LIN {X 0,Y 312.695,Z 496.66,A -85,B 0,C 180,E1 -15735.686,E2 -15735.686} C_VEL
LIN {X 0,Y 312.703,Z 496.659,A -85,B 0,C 180,E1 -15739.642,E2 -15739.642} C_VEL
LIN {X 0,Y 312.873,Z 496.634,A -85,B 0,C 180,E1 -15742.254,E2 -15742.254} C_VEL
LIN {X 0,Y 312.72,Z 496.654,A -85,B 0,C 180,E1 -15744.842,E2 -15744.842} C_VEL
LIN {X 0,Y 312.954,Z 496.629,A -85,B 0,C 180,E1 -15747.426,E2 -15747.426} C_VEL
LIN {X 0,Y 313.122,Z 496.604,A -85,B 0,C 180,E1 -15750,E2 -15750} C_VEL
LIN {X 0,Y 312.94,Z 496.626,A -85,B 0,C 180,E1 -15752.574,E2 -15752.574} C_VEL
LIN {X 0,Y 312.911,Z 496.629,A -85,B 0,C 180,E1 -15756.448,E2 -15756.448} C_VEL
LIN {X 0,Y 312.789,Z 496.646,A -85,B 0,C 180,E1 -15759.049,E2 -15759.049} C_VEL
LIN {X 0,Y 312.636,Z 496.666,A -85,B 0,C 180,E1 -15762.991,E2 -15762.991} C_VEL
LIN {X 0,Y 312.639,Z 496.666,A -85,B 0,C 180,E1 -15765.65,E2 -15765.65} C_VEL
LIN {X 0,Y 312.631,Z 496.668,A -85,B 0,C 180,E1 -15769.237,E2 -15769.237} C_VEL
LIN {X 0,Y 312.547,Z 496.676,A -85,B 0,C 180,E1 -15772.789,E2 -15772.789} C_VEL
LIN {X 0,Y 312.598,Z 496.669,A -85,B 0,C 180,E1 -15775.933,E2 -15775.933} C_VEL
LIN {X 0,Y 312.539,Z 496.679,A -85,B 0,C 180,E1 -15779.651,E2 -15779.651} C_VEL
LIN {X 0,Y 312.52,Z 496.68,A -85,B 0,C 180,E1 -15783.689,E2 -15783.689} C_VEL
LIN {X 0,Y 312.539,Z 496.681,A -85,B 0,C 180,E1 -15787.383,E2 -15787.383} C_VEL
LIN {X 0,Y 312.491,Z 496.682,A -85,B 0,C 180,E1 -15790.709,E2 -15790.709} C_VEL
LIN {X 0,Y 312.473,Z 496.684,A -85,B 0,C 180,E1 -15794.206,E2 -15794.206} C_VEL
LIN {X 0,Y 312.487,Z 496.683,A -85,B 0,C 180,E1 -15797.918,E2 -15797.918} C_VEL
LIN {X 0,Y 312.507,Z 496.681,A -85,B 0,C 180,E1 -15801.917,E2 -15801.917} C_VEL
LIN {X 0,Y 312.533,Z 496.677,A -85,B 0,C 180,E1 -15804.22,E2 -15804.22} C_VEL
LIN {X 0,Y 312.548,Z 496.702,A -85,B 0,C 180,E1 -15806.423,E2 -15806.423} C_VEL
LIN {X 0,Y 316.105,Z 512.177,A -85,B 0,C 180,E1 -15809.735,E2 -15809.735} C_VEL
LIN {X 0,Y 318.578,Z 524.112,A -85,B 0,C 180,E1 -15812.214,E2 -15812.214} C_VEL
LIN {X 0,Y 317.779,Z 535.92,A -85,B 0,C 180,E1 -15814.452,E2 -15814.452} C_VEL
LIN {X 0,Y 317.727,Z 536.622,A -85,B 0,C 180,E1 -15814.586,E2 -15814.586} C_VEL
LIN {X 0,Y 316.838,Z 539.658,A -85,B 0,C 180,E1 -15815.123,E2 -15815.123} C_VEL
LIN {X 0,Y 313.587,Z 544.619,A -85,B 0,C 180,E1 -15815.91,E2 -15815.91} C_VEL
LIN {X 0,Y 310.704,Z 549.223,A -85,B 0,C 180,E1 -15816.517,E2 -15816.517} C_VEL
LIN {X 0,Y 310.133,Z 552.013,A -85,B 0,C 180,E1 -15816.724,E2 -15816.724} C_VEL
LIN {X 0,Y 310.154,Z 552.609,A -85,B 0,C 180,E1 -15816.751,E2 -15816.751} C_VEL
LIN {X 0,Y 313.108,Z 577.851,A -85,B 0,C 180,E1 -15817.752,E2 -15817.752} C_VEL
LIN {X 0,Y 310.286,Z 660.865,A -85,B 0,C 180,E1 -15820.483,E2 -15820.483} C_VEL
LIN {X 0,Y 309.628,Z 673.725,A -85,B 0,C 180,E1 -15821.128,E2 -15821.128} C_VEL
LIN {X 0,Y 308.833,Z 687.47,A -85,B 0,C 180,E1 -15822.109,E2 -15822.109} C_VEL
LIN {X 0,Y 308,Z 699.244,A -85,B 0,C 180,E1 -15823.207,E2 -15823.207} C_VEL
LIN {X 0,Y 307.266,Z 709.548,A -85,B 0,C 180,E1 -15824.41,E2 -15824.41} C_VEL
LIN {X 0,Y 306.424,Z 719.942,A -85,B 0,C 180,E1 -15825.896,E2 -15825.896} C_VEL
LIN {X 0,Y 305.623,Z 728.532,A -85,B 0,C 180,E1 -15827.381,E2 -15827.381} C_VEL
LIN {X 0,Y 304.853,Z 737.882,A -85,B 0,C 180,E1 -15829.372,E2 -15829.372} C_VEL
LIN {X 0,Y 304.29,Z 745.423,A -85,B 0,C 180,E1 -15831.366,E2 -15831.366} C_VEL
LIN {X 0,Y 303.987,Z 751.404,A -85,B 0,C 180,E1 -15833.362,E2 -15833.362} C_VEL
LIN {X 0,Y 303.777,Z 756.071,A -85,B 0,C 180,E1 -15835.355,E2 -15835.355} C_VEL
LIN {X 0,Y 303.663,Z 759.57,A -85,B 0,C 180,E1 -15837.347,E2 -15837.347} C_VEL
LIN {X 0,Y 303.58,Z 761.313,A -85,B 0,C 180,E1 -15838.673,E2 -15838.673} C_VEL
LIN {X 0,Y 303.601,Z 762.593,A -85,B 0,C 180,E1 -15840,E2 -15840} C_VEL
LIN {X 0,Y 303.634,Z 763.4,A -85,B 0,C 180,E1 -15841.326,E2 -15841.326} C_VEL
LIN {X 0,Y 303.73,Z 763.791,A -85,B 0,C 180,E1 -15842.653,E2 -15842.653} C_VEL
LIN {X 0,Y 303.896,Z 763.755,A -85,B 0,C 180,E1 -15843.978,E2 -15843.978} C_VEL
LIN {X 0,Y 304.174,Z 763.245,A -85,B 0,C 180,E1 -15845.303,E2 -15845.303} C_VEL
LIN {X 0,Y 304.765,Z 761.541,A -85,B 0,C 180,E1 -15847.432,E2 -15847.432} C_VEL
LIN {X 0,Y 305.648,Z 758.098,A -85,B 0,C 180,E1 -15849.931,E2 -15849.931} C_VEL
LIN {X 0,Y 306.73,Z 754.162,A -85,B 0,C 180,E1 -15851.901,E2 -15851.901} C_VEL
LIN {X 0,Y 308.02,Z 749.044,A -85,B 0,C 180,E1 -15853.862,E2 -15853.862} C_VEL
LIN {X 0,Y 309.69,Z 742.568,A -85,B 0,C 180,E1 -15855.803,E2 -15855.803} C_VEL
LIN {X 0,Y 311.786,Z 734.624,A -85,B 0,C 180,E1 -15857.716,E2 -15857.716} C_VEL
LIN {X 0,Y 313.755,Z 726.562,A -85,B 0,C 180,E1 -15859.293,E2 -15859.293} C_VEL
LIN {X 0,Y 316.124,Z 715.871,A -85,B 0,C 180,E1 -15860.975,E2 -15860.975} C_VEL
LIN {X 0,Y 318.27,Z 704.858,A -85,B 0,C 180,E1 -15862.39,E2 -15862.39} C_VEL
LIN {X 0,Y 320.467,Z 692.846,A -85,B 0,C 180,E1 -15863.593,E2 -15863.593} C_VEL
LIN {X 0,Y 322.376,Z 680.473,A -85,B 0,C 180,E1 -15864.556,E2 -15864.556} C_VEL
LIN {X 0,Y 324.061,Z 666.63,A -85,B 0,C 180,E1 -15865.361,E2 -15865.361} C_VEL
LIN {X 0,Y 326.296,Z 642.291,A -85,B 0,C 180,E1 -15866.332,E2 -15866.332} C_VEL
LIN {X 0,Y 332.02,Z 585.244,A -85,B 0,C 180,E1 -15868.52,E2 -15868.52} C_VEL
LIN {X 0,Y 330.422,Z 572.445,A -85,B 0,C 180,E1 -15869.651,E2 -15869.651} C_VEL
LIN {X 0,Y 328.053,Z 558.26,A -85,B 0,C 180,E1 -15871.202,E2 -15871.202} C_VEL
LIN {X 0,Y 327.111,Z 552.951,A -85,B 0,C 180,E1 -15871.875,E2 -15871.875} C_VEL
LIN {X 0,Y 326.796,Z 547.751,A -85,B 0,C 180,E1 -15873.522,E2 -15873.522} C_VEL
LIN {X 0,Y 326.075,Z 542.207,A -85,B 0,C 180,E1 -15875.587,E2 -15875.587} C_VEL
LIN {X 0,Y 325.136,Z 537.325,A -85,B 0,C 180,E1 -15877.875,E2 -15877.875} C_VEL
LIN {X 0,Y 324.526,Z 534.263,A -85,B 0,C 180,E1 -15879.638,E2 -15879.638} C_VEL
LIN {X 0,Y 323.75,Z 531.075,A -85,B 0,C 180,E1 -15882.295,E2 -15882.295} C_VEL
LIN {X 0,Y 323.483,Z 529.687,A -85,B 0,C 180,E1 -15884.196,E2 -15884.196} C_VEL
LIN {X 0,Y 323.536,Z 529.08,A -85,B 0,C 180,E1 -15885.963,E2 -15885.963} C_VEL
LIN {X 0,Y 323.915,Z 529.107,A -85,B 0,C 180,E1 -15887.731,E2 -15887.731} C_VEL
LIN {X 0,Y 324.623,Z 529.847,A -85,B 0,C 180,E1 -15889.497,E2 -15889.497} C_VEL
LIN {X 0,Y 325.763,Z 531.237,A -85,B 0,C 180,E1 -15891.27,E2 -15891.27} C_VEL
LIN {X 0,Y 327.409,Z 533.393,A -85,B 0,C 180,E1 -15893.056,E2 -15893.056} C_VEL
LIN {X 0,Y 329.137,Z 536.699,A -85,B 0,C 180,E1 -15894.793,E2 -15894.793} C_VEL
LIN {X 0,Y 329.649,Z 540.65,A -85,B 0,C 180,E1 -15895.886,E2 -15895.886} C_VEL
LIN {X 0,Y 330.931,Z 549.612,A -85,B 0,C 180,E1 -15897.932,E2 -15897.932} C_VEL
LIN {X 0,Y 331.047,Z 551.894,A -85,B 0,C 180,E1 -15898.332,E2 -15898.332} C_VEL
LIN {X 0,Y 330.217,Z 558.252,A -85,B 0,C 180,E1 -15899.044,E2 -15899.044} C_VEL
LIN {X 0,Y 330.357,Z 566.805,A -85,B 0,C 180,E1 -15899.668,E2 -15899.668} C_VEL
LIN {X 0,Y 321.228,Z 657.87,A -85,B 0,C 180,E1 -15903.396,E2 -15903.396} C_VEL
LIN {X 0,Y 319.332,Z 680.325,A -85,B 0,C 180,E1 -15904.367,E2 -15904.367} C_VEL
LIN {X 0,Y 317.783,Z 694.511,A -85,B 0,C 180,E1 -15905.267,E2 -15905.267} C_VEL
LIN {X 0,Y 316.222,Z 706.55,A -85,B 0,C 180,E1 -15906.266,E2 -15906.266} C_VEL
LIN {X 0,Y 314.48,Z 718.218,A -85,B 0,C 180,E1 -15907.498,E2 -15907.498} C_VEL
LIN {X 0,Y 312.297,Z 730.334,A -85,B 0,C 180,E1 -15909.068,E2 -15909.068} C_VEL
LIN {X 0,Y 310.283,Z 741.053,A -85,B 0,C 180,E1 -15910.826,E2 -15910.826} C_VEL
LIN {X 0,Y 308.438,Z 750.629,A -85,B 0,C 180,E1 -15912.77,E2 -15912.77} C_VEL
LIN {X 0,Y 306.979,Z 758.385,A -85,B 0,C 180,E1 -15914.735,E2 -15914.735} C_VEL
LIN {X 0,Y 305.773,Z 764.7,A -85,B 0,C 180,E1 -15916.712,E2 -15916.712} C_VEL
LIN {X 0,Y 304.895,Z 769.78,A -85,B 0,C 180,E1 -15918.701,E2 -15918.701} C_VEL
LIN {X 0,Y 304.243,Z 773.698,A -85,B 0,C 180,E1 -15920.694,E2 -15920.694} C_VEL
LIN {X 0,Y 303.964,Z 775.739,A -85,B 0,C 180,E1 -15922.026,E2 -15922.026} C_VEL
LIN {X 0,Y 303.689,Z 778.175,A -85,B 0,C 180,E1 -15924.332,E2 -15924.332} C_VEL
LIN {X 0,Y 303.601,Z 779.137,A -85,B 0,C 180,E1 -15926.018,E2 -15926.018} C_VEL
LIN {X 0,Y 303.627,Z 779.384,A -85,B 0,C 180,E1 -15927.347,E2 -15927.347} C_VEL
LIN {X 0,Y 303.622,Z 779.172,A -85,B 0,C 180,E1 -15928.674,E2 -15928.674} C_VEL
LIN {X 0,Y 303.591,Z 780.184,A -85,B 0,C 180,E1 -15931.327,E2 -15931.327} C_VEL
LIN {X 0,Y 303.608,Z 780.324,A -85,B 0,C 180,E1 -15932.654,E2 -15932.654} C_VEL
LIN {X 0,Y 303.617,Z 779.456,A -85,B 0,C 180,E1 -15935.313,E2 -15935.313} C_VEL
LIN {X 0,Y 303.931,Z 777.116,A -85,B 0,C 180,E1 -15937.975,E2 -15937.975} C_VEL
LIN {X 0,Y 304.585,Z 773.291,A -85,B 0,C 180,E1 -15940.638,E2 -15940.638} C_VEL
LIN {X 0,Y 305.761,Z 767.896,A -85,B 0,C 180,E1 -15943.289,E2 -15943.289} C_VEL
LIN {X 0,Y 306.969,Z 762.706,A -85,B 0,C 180,E1 -15945.266,E2 -15945.266} C_VEL
LIN {X 0,Y 308.805,Z 755.301,A -85,B 0,C 180,E1 -15947.551,E2 -15947.551} C_VEL
LIN {X 0,Y 311.045,Z 746.197,A -85,B 0,C 180,E1 -15949.811,E2 -15949.811} C_VEL
LIN {X 0,Y 313.455,Z 736.695,A -85,B 0,C 180,E1 -15951.713,E2 -15951.713} C_VEL
LIN {X 0,Y 316.278,Z 725.263,A -85,B 0,C 180,E1 -15953.577,E2 -15953.577} C_VEL
LIN {X 0,Y 318.903,Z 713.895,A -85,B 0,C 180,E1 -15955.088,E2 -15955.088} C_VEL
LIN {X 0,Y 321.678,Z 700.835,A -85,B 0,C 180,E1 -15956.481,E2 -15956.481} C_VEL
LIN {X 0,Y 324.109,Z 687.483,A -85,B 0,C 180,E1 -15957.613,E2 -15957.613} C_VEL
LIN {X 0,Y 326.649,Z 671.83,A -85,B 0,C 180,E1 -15958.602,E2 -15958.602} C_VEL
LIN {X 0,Y 328.391,Z 657.161,A -85,B 0,C 180,E1 -15959.268,E2 -15959.268} C_VEL
LIN {X 0,Y 335.537,Z 586.231,A -85,B 0,C 180,E1 -15961.806,E2 -15961.806} C_VEL
LIN {X 0,Y 337.662,Z 566.7,A -85,B 0,C 180,E1 -15962.538,E2 -15962.538} C_VEL
LIN {X 0,Y 337.163,Z 562,A -85,B 0,C 180,E1 -15962.964,E2 -15962.964} C_VEL
LIN {X 0,Y 334.12,Z 555.825,A -85,B 0,C 180,E1 -15964.156,E2 -15964.156} C_VEL
LIN {X 0,Y 331.829,Z 551.509,A -85,B 0,C 180,E1 -15965.145,E2 -15965.145} C_VEL
LIN {X 0,Y 329.918,Z 548.193,A -85,B 0,C 180,E1 -15966.033,E2 -15966.033} C_VEL
LIN {X 0,Y 327.363,Z 544.086,A -85,B 0,C 180,E1 -15967.336,E2 -15967.336} C_VEL
LIN {X 0,Y 323.847,Z 539.068,A -85,B 0,C 180,E1 -15969.498,E2 -15969.498} C_VEL
LIN {X 0,Y 320.513,Z 534.919,A -85,B 0,C 180,E1 -15972.459,E2 -15972.459} C_VEL
LIN {X 0,Y 319.82,Z 533.854,A -85,B 0,C 180,E1 -15973.517,E2 -15973.517} C_VEL
LIN {X 0,Y 319.684,Z 533.495,A -85,B 0,C 180,E1 -15976.509,E2 -15976.509} C_VEL
LIN {X 0,Y 319.826,Z 534.162,A -85,B 0,C 180,E1 -15978.759,E2 -15978.759} C_VEL
LIN {X 0,Y 320.214,Z 535.661,A -85,B 0,C 180,E1 -15980.843,E2 -15980.843} C_VEL
LIN {X 0,Y 323.301,Z 540.989,A -85,B 0,C 180,E1 -15983.922,E2 -15983.922} C_VEL
LIN {X 0,Y 324.67,Z 543.01,A -85,B 0,C 180,E1 -15984.879,E2 -15984.879} C_VEL
LIN {X 0,Y 328.101,Z 549.368,A -85,B 0,C 180,E1 -15986.957,E2 -15986.957} C_VEL
LIN {X 0,Y 330.938,Z 555.184,A -85,B 0,C 180,E1 -15988.434,E2 -15988.434} C_VEL
LIN {X 0,Y 332.724,Z 559.305,A -85,B 0,C 180,E1 -15989.287,E2 -15989.287} C_VEL
LIN {X 0,Y 334.38,Z 571.019,A -85,B 0,C 180,E1 -15990.609,E2 -15990.609} C_VEL
LIN {X 0,Y 335.309,Z 581.125,A -85,B 0,C 180,E1 -15991.553,E2 -15991.553} C_VEL
LIN {X 0,Y 335.436,Z 584.56,A -85,B 0,C 180,E1 -15991.807,E2 -15991.807} C_VEL
LIN {X 0,Y 326.755,Z 659.896,A -85,B 0,C 180,E1 -15994.864,E2 -15994.864} C_VEL
LIN {X 0,Y 324.963,Z 672.654,A -85,B 0,C 180,E1 -15995.61,E2 -15995.61} C_VEL
LIN {X 0,Y 322.419,Z 687.269,A -85,B 0,C 180,E1 -15996.747,E2 -15996.747} C_VEL
LIN {X 0,Y 320.224,Z 699.057,A -85,B 0,C 180,E1 -15997.923,E2 -15997.923} C_VEL
LIN {X 0,Y 317.517,Z 711.185,A -85,B 0,C 180,E1 -15999.428,E2 -15999.428} C_VEL
LIN {X 0,Y 314.904,Z 722.101,A -85,B 0,C 180,E1 -16001.119,E2 -16001.119} C_VEL
LIN {X 0,Y 312.39,Z 731.847,A -85,B 0,C 180,E1 -16002.994,E2 -16002.994} C_VEL
LIN {X 0,Y 310.347,Z 739.777,A -85,B 0,C 180,E1 -16004.905,E2 -16004.905} C_VEL
LIN {X 0,Y 308.598,Z 746.288,A -85,B 0,C 180,E1 -16006.836,E2 -16006.836} C_VEL
LIN {X 0,Y 307.089,Z 751.53,A -85,B 0,C 180,E1 -16008.783,E2 -16008.783} C_VEL
LIN {X 0,Y 305.999,Z 755.591,A -85,B 0,C 180,E1 -16010.748,E2 -16010.748} C_VEL
LIN {X 0,Y 305.368,Z 757.72,A -85,B 0,C 180,E1 -16012.063,E2 -16012.063} C_VEL
LIN {X 0,Y 304.764,Z 759.412,A -85,B 0,C 180,E1 -16013.379,E2 -16013.379} C_VEL
LIN {X 0,Y 304.373,Z 760.671,A -85,B 0,C 180,E1 -16014.701,E2 -16014.701} C_VEL
LIN {X 0,Y 304.136,Z 761.512,A -85,B 0,C 180,E1 -16016.025,E2 -16016.025} C_VEL
LIN {X 0,Y 303.912,Z 761.908,A -85,B 0,C 180,E1 -16017.349,E2 -16017.349} C_VEL
LIN {X 0,Y 303.732,Z 761.869,A -85,B 0,C 180,E1 -16018.674,E2 -16018.674} C_VEL
LIN {X 0,Y 303.639,Z 761.416,A -85,B 0,C 180,E1 -16020,E2 -16020} C_VEL
LIN {X 0,Y 303.615,Z 760.545,A -85,B 0,C 180,E1 -16021.326,E2 -16021.326} C_VEL
LIN {X 0,Y 303.658,Z 759.214,A -85,B 0,C 180,E1 -16022.653,E2 -16022.653} C_VEL
LIN {X 0,Y 303.667,Z 756.37,A -85,B 0,C 180,E1 -16024.646,E2 -16024.646} C_VEL
LIN {X 0,Y 303.858,Z 752.437,A -85,B 0,C 180,E1 -16026.641,E2 -16026.641} C_VEL
LIN {X 0,Y 304.142,Z 747.299,A -85,B 0,C 180,E1 -16028.638,E2 -16028.638} C_VEL
LIN {X 0,Y 304.695,Z 739.609,A -85,B 0,C 180,E1 -16030.97,E2 -16030.97} C_VEL
LIN {X 0,Y 305.417,Z 731.304,A -85,B 0,C 180,E1 -16032.965,E2 -16032.965} C_VEL
LIN {X 0,Y 306.216,Z 721.523,A -85,B 0,C 180,E1 -16034.853,E2 -16034.853} C_VEL
LIN {X 0,Y 307.126,Z 711.43,A -85,B 0,C 180,E1 -16036.45,E2 -16036.45} C_VEL
LIN {X 0,Y 308.19,Z 699.881,A -85,B 0,C 180,E1 -16037.93,E2 -16037.93} C_VEL
LIN {X 0,Y 309.268,Z 687.138,A -85,B 0,C 180,E1 -16039.239,E2 -16039.239} C_VEL
LIN {X 0,Y 310.192,Z 673.757,A -85,B 0,C 180,E1 -16040.3,E2 -16040.3} C_VEL
LIN {X 0,Y 311.018,Z 659.239,A -85,B 0,C 180,E1 -16041.152,E2 -16041.152} C_VEL
LIN {X 0,Y 311.791,Z 641.246,A -85,B 0,C 180,E1 -16041.834,E2 -16041.834} C_VEL
LIN {X 0,Y 314.384,Z 574.76,A -85,B 0,C 180,E1 -16044.078,E2 -16044.078} C_VEL
LIN {X 0,Y 310.271,Z 540.944,A -85,B 0,C 180,E1 -16045.514,E2 -16045.514} C_VEL
LIN {X 0,Y 310.116,Z 539.007,A -85,B 0,C 180,E1 -16045.595,E2 -16045.595} C_VEL
LIN {X 0,Y 311.695,Z 526.352,A -85,B 0,C 180,E1 -16048.628,E2 -16048.628} C_VEL
LIN {X 0,Y 309.2,Z 514.335,A -85,B 0,C 180,E1 -16051.833,E2 -16051.833} C_VEL
LIN {X 0,Y 306.408,Z 501.538,A -85,B 0,C 180,E1 -16055.391,E2 -16055.391} C_VEL
LIN {X 0,Y 305.508,Z 497.552,A -85,B 0,C 180,E1 -16056.557,E2 -16056.557} C_VEL
LIN {X 0,Y 305.46,Z 497.558,A -85,B 0,C 180,E1 -16060.107,E2 -16060.107} C_VEL
LIN {X 0,Y 305.43,Z 497.566,A -85,B 0,C 180,E1 -16063.654,E2 -16063.654} C_VEL
LIN {X 0,Y 305.456,Z 497.562,A -85,B 0,C 180,E1 -16067.414,E2 -16067.414} C_VEL
LIN {X 0,Y 305.477,Z 497.561,A -85,B 0,C 180,E1 -16071.597,E2 -16071.597} C_VEL
LIN {X 0,Y 305.464,Z 497.557,A -85,B 0,C 180,E1 -16074.887,E2 -16074.887} C_VEL
LIN {X 0,Y 305.454,Z 497.558,A -85,B 0,C 180,E1 -16078.354,E2 -16078.354} C_VEL
LIN {X 0,Y 305.522,Z 497.552,A -85,B 0,C 180,E1 -16081.114,E2 -16081.114} C_VEL
LIN {X 0,Y 305.573,Z 497.544,A -85,B 0,C 180,E1 -16084.088,E2 -16084.088} C_VEL
LIN {X 0,Y 305.503,Z 497.552,A -85,B 0,C 180,E1 -16088.403,E2 -16088.403} C_VEL
LIN {X 0,Y 305.592,Z 497.544,A -85,B 0,C 180,E1 -16091.218,E2 -16091.218} C_VEL
LIN {X 0,Y 305.65,Z 497.538,A -85,B 0,C 180,E1 -16095.349,E2 -16095.349} C_VEL
LIN {X 0,Y 305.64,Z 497.54,A -85,B 0,C 180,E1 -16099.4,E2 -16099.4} C_VEL
LIN {X 0,Y 305.814,Z 497.514,A -85,B 0,C 180,E1 -16102.074,E2 -16102.074} C_VEL
LIN {X 0,Y 305.692,Z 497.529,A -85,B 0,C 180,E1 -16104.723,E2 -16104.723} C_VEL
LIN {X 0,Y 305.961,Z 497.495,A -85,B 0,C 180,E1 -16108.684,E2 -16108.684} C_VEL
LIN {X 0,Y 305.959,Z 497.499,A -85,B 0,C 180,E1 -16111.316,E2 -16111.316} C_VEL
LIN {X 0,Y 305.853,Z 497.508,A -85,B 0,C 180,E1 -16116.597,E2 -16116.597} C_VEL
LIN {X 0,Y 305.737,Z 497.526,A -85,B 0,C 180,E1 -16119.26,E2 -16119.26} C_VEL
LIN {X 0,Y 305.591,Z 497.546,A -85,B 0,C 180,E1 -16123.296,E2 -16123.296} C_VEL
LIN {X 0,Y 305.595,Z 497.541,A -85,B 0,C 180,E1 -16126.02,E2 -16126.02} C_VEL
LIN {X 0,Y 305.578,Z 497.548,A -85,B 0,C 180,E1 -16129.445,E2 -16129.445} C_VEL
LIN {X 0,Y 305.492,Z 497.556,A -85,B 0,C 180,E1 -16133.042,E2 -16133.042} C_VEL
LIN {X 0,Y 305.527,Z 497.549,A -85,B 0,C 180,E1 -16136.219,E2 -16136.219} C_VEL
LIN {X 0,Y 305.489,Z 497.557,A -85,B 0,C 180,E1 -16139.047,E2 -16139.047} C_VEL
LIN {X 0,Y 305.443,Z 497.56,A -85,B 0,C 180,E1 -16141.952,E2 -16141.952} C_VEL
LIN {X 0,Y 305.464,Z 497.56,A -85,B 0,C 180,E1 -16145.113,E2 -16145.113} C_VEL
LIN {X 0,Y 305.468,Z 497.557,A -85,B 0,C 180,E1 -16148.533,E2 -16148.533} C_VEL
LIN {X 0,Y 305.46,Z 497.557,A -85,B 0,C 180,E1 -16152.587,E2 -16152.587} C_VEL
LIN {X 0,Y 305.444,Z 497.559,A -85,B 0,C 180,E1 -16156.348,E2 -16156.348} C_VEL
LIN {X 0,Y 305.459,Z 497.559,A -85,B 0,C 180,E1 -16159.892,E2 -16159.892} C_VEL
LIN {X 0,Y 305.482,Z 497.558,A -85,B 0,C 180,E1 -16163.632,E2 -16163.632} C_VEL
LIN {X 0,Y 305.504,Z 497.666,A -85,B 0,C 180,E1 -16166.1,E2 -16166.1} C_VEL
LIN {X 0,Y 309.184,Z 513.586,A -85,B 0,C 180,E1 -16169.557,E2 -16169.557} C_VEL
LIN {X 0,Y 311.742,Z 526.155,A -85,B 0,C 180,E1 -16172.209,E2 -16172.209} C_VEL
LIN {X 0,Y 309.916,Z 549.112,A -85,B 0,C 180,E1 -16176.592,E2 -16176.592} C_VEL
LIN {X 0,Y 310.154,Z 552.609,A -85,B 0,C 180,E1 -16176.751,E2 -16176.751} C_VEL
LIN {X 0,Y 310.121,Z 558.432,A -85,B 0,C 180,E1 -16176.95,E2 -16176.95} C_VEL
LIN {X 0,Y 308.576,Z 568.1,A -85,B 0,C 180,E1 -16177.22,E2 -16177.22} C_VEL
LIN {X 0,Y 306.969,Z 575.849,A -85,B 0,C 180,E1 -16177.422,E2 -16177.422} C_VEL
LIN {X 0,Y 305.977,Z 583.656,A -85,B 0,C 180,E1 -16177.651,E2 -16177.651} C_VEL
LIN {X 0,Y 303.278,Z 660.661,A -85,B 0,C 180,E1 -16180.278,E2 -16180.278} C_VEL
LIN {X 0,Y 302.616,Z 673.524,A -85,B 0,C 180,E1 -16180.938,E2 -16180.938} C_VEL
LIN {X 0,Y 301.793,Z 687.269,A -85,B 0,C 180,E1 -16181.94,E2 -16181.94} C_VEL
LIN {X 0,Y 300.945,Z 699.391,A -85,B 0,C 180,E1 -16183.097,E2 -16183.097} C_VEL
LIN {X 0,Y 300.24,Z 708.783,A -85,B 0,C 180,E1 -16184.21,E2 -16184.21} C_VEL
LIN {X 0,Y 299.384,Z 719.33,A -85,B 0,C 180,E1 -16185.73,E2 -16185.73} C_VEL
LIN {X 0,Y 298.512,Z 728.964,A -85,B 0,C 180,E1 -16187.422,E2 -16187.422} C_VEL
LIN {X 0,Y 297.724,Z 738.281,A -85,B 0,C 180,E1 -16189.459,E2 -16189.459} C_VEL
LIN {X 0,Y 297.162,Z 745.8,A -85,B 0,C 180,E1 -16191.5,E2 -16191.5} C_VEL
LIN {X 0,Y 296.863,Z 751.947,A -85,B 0,C 180,E1 -16193.62,E2 -16193.62} C_VEL
LIN {X 0,Y 296.672,Z 757.075,A -85,B 0,C 180,E1 -16195.925,E2 -16195.925} C_VEL
LIN {X 0,Y 296.593,Z 759.387,A -85,B 0,C 180,E1 -16197.284,E2 -16197.284} C_VEL
LIN {X 0,Y 296.501,Z 761.194,A -85,B 0,C 180,E1 -16198.642,E2 -16198.642} C_VEL
LIN {X 0,Y 296.516,Z 762.576,A -85,B 0,C 180,E1 -16200,E2 -16200} C_VEL
LIN {X 0,Y 296.552,Z 763.5,A -85,B 0,C 180,E1 -16201.358,E2 -16201.358} C_VEL
LIN {X 0,Y 296.657,Z 763.969,A -85,B 0,C 180,E1 -16202.716,E2 -16202.716} C_VEL
LIN {X 0,Y 296.841,Z 764.025,A -85,B 0,C 180,E1 -16204.073,E2 -16204.073} C_VEL
LIN {X 0,Y 297.12,Z 763.647,A -85,B 0,C 180,E1 -16205.429,E2 -16205.429} C_VEL
LIN {X 0,Y 297.707,Z 762.238,A -85,B 0,C 180,E1 -16207.475,E2 -16207.475} C_VEL
LIN {X 0,Y 298.698,Z 758.856,A -85,B 0,C 180,E1 -16210.164,E2 -16210.164} C_VEL
LIN {X 0,Y 299.851,Z 755.084,A -85,B 0,C 180,E1 -16212.178,E2 -16212.178} C_VEL
LIN {X 0,Y 301.227,Z 750.184,A -85,B 0,C 180,E1 -16214.181,E2 -16214.181} C_VEL
LIN {X 0,Y 303.018,Z 744.027,A -85,B 0,C 180,E1 -16216.16,E2 -16216.16} C_VEL
LIN {X 0,Y 305.22,Z 736.308,A -85,B 0,C 180,E1 -16218.111,E2 -16218.111} C_VEL
LIN {X 0,Y 307.728,Z 726.835,A -85,B 0,C 180,E1 -16220.034,E2 -16220.034} C_VEL
LIN {X 0,Y 310.104,Z 717.108,A -85,B 0,C 180,E1 -16221.618,E2 -16221.618} C_VEL
LIN {X 0,Y 312.299,Z 706.644,A -85,B 0,C 180,E1 -16223.017,E2 -16223.017} C_VEL
LIN {X 0,Y 314.615,Z 695.046,A -85,B 0,C 180,E1 -16224.234,E2 -16224.234} C_VEL
LIN {X 0,Y 316.762,Z 682.47,A -85,B 0,C 180,E1 -16225.284,E2 -16225.284} C_VEL
LIN {X 0,Y 318.58,Z 669.417,A -85,B 0,C 180,E1 -16226.093,E2 -16226.093} C_VEL
LIN {X 0,Y 320.019,Z 655.52,A -85,B 0,C 180,E1 -16226.713,E2 -16226.713} C_VEL
LIN {X 0,Y 327.311,Z 587.133,A -85,B 0,C 180,E1 -16229.393,E2 -16229.393} C_VEL
LIN {X 0,Y 326.04,Z 575.187,A -85,B 0,C 180,E1 -16230.509,E2 -16230.509} C_VEL
LIN {X 0,Y 324.082,Z 561.884,A -85,B 0,C 180,E1 -16232.016,E2 -16232.016} C_VEL
LIN {X 0,Y 323.145,Z 557.029,A -85,B 0,C 180,E1 -16232.682,E2 -16232.682} C_VEL
LIN {X 0,Y 321.748,Z 553.348,A -85,B 0,C 180,E1 -16233.473,E2 -16233.473} C_VEL
LIN {X 0,Y 321.154,Z 546.931,A -85,B 0,C 180,E1 -16235.934,E2 -16235.934} C_VEL
LIN {X 0,Y 320.509,Z 542.896,A -85,B 0,C 180,E1 -16237.877,E2 -16237.877} C_VEL
LIN {X 0,Y 320.034,Z 539.727,A -85,B 0,C 180,E1 -16239.771,E2 -16239.771} C_VEL
LIN {X 0,Y 319.55,Z 537.494,A -85,B 0,C 180,E1 -16241.602,E2 -16241.602} C_VEL
LIN {X 0,Y 319.342,Z 535.956,A -85,B 0,C 180,E1 -16243.426,E2 -16243.426} C_VEL
LIN {X 0,Y 319.367,Z 535.105,A -85,B 0,C 180,E1 -16245.235,E2 -16245.235} C_VEL
LIN {X 0,Y 319.727,Z 534.921,A -85,B 0,C 180,E1 -16247.045,E2 -16247.045} C_VEL
LIN {X 0,Y 320.388,Z 535.452,A -85,B 0,C 180,E1 -16248.846,E2 -16248.846} C_VEL
LIN {X 0,Y 322.323,Z 537.729,A -85,B 0,C 180,E1 -16251.716,E2 -16251.716} C_VEL
LIN {X 0,Y 323.052,Z 538.562,A -85,B 0,C 180,E1 -16252.473,E2 -16252.473} C_VEL
LIN {X 0,Y 324.824,Z 541.722,A -85,B 0,C 180,E1 -16254.255,E2 -16254.255} C_VEL
LIN {X 0,Y 325.11,Z 542.715,A -85,B 0,C 180,E1 -16254.639,E2 -16254.639} C_VEL
LIN {X 0,Y 326.062,Z 551.664,A -85,B 0,C 180,E1 -16256.864,E2 -16256.864} C_VEL
LIN {X 0,Y 326.393,Z 555.481,A -85,B 0,C 180,E1 -16257.629,E2 -16257.629} C_VEL
LIN {X 0,Y 326.023,Z 559.073,A -85,B 0,C 180,E1 -16258.007,E2 -16258.007} C_VEL
LIN {X 0,Y 326.11,Z 567.867,A -85,B 0,C 180,E1 -16258.693,E2 -16258.693} C_VEL
LIN {X 0,Y 316.411,Z 656.598,A -85,B 0,C 180,E1 -16262.421,E2 -16262.421} C_VEL
LIN {X 0,Y 314.18,Z 680.026,A -85,B 0,C 180,E1 -16263.468,E2 -16263.468} C_VEL
LIN {X 0,Y 312.61,Z 692.853,A -85,B 0,C 180,E1 -16264.267,E2 -16264.267} C_VEL
LIN {X 0,Y 310.671,Z 706.419,A -85,B 0,C 180,E1 -16265.412,E2 -16265.412} C_VEL
LIN {X 0,Y 308.474,Z 719.6,A -85,B 0,C 180,E1 -16266.858,E2 -16266.858} C_VEL
LIN {X 0,Y 306.36,Z 730.271,A -85,B 0,C 180,E1 -16268.29,E2 -16268.29} C_VEL
LIN {X 0,Y 304.109,Z 740.872,A -85,B 0,C 180,E1 -16270.07,E2 -16270.07} C_VEL
LIN {X 0,Y 302.044,Z 750.416,A -85,B 0,C 180,E1 -16272.043,E2 -16272.043} C_VEL
LIN {X 0,Y 300.189,Z 759.254,A -85,B 0,C 180,E1 -16274.381,E2 -16274.381} C_VEL
LIN {X 0,Y 298.889,Z 765.379,A -85,B 0,C 180,E1 -16276.4,E2 -16276.4} C_VEL
LIN {X 0,Y 297.924,Z 770.231,A -85,B 0,C 180,E1 -16278.433,E2 -16278.433} C_VEL
LIN {X 0,Y 297.216,Z 773.98,A -85,B 0,C 180,E1 -16280.472,E2 -16280.472} C_VEL
LIN {X 0,Y 296.919,Z 775.878,A -85,B 0,C 180,E1 -16281.835,E2 -16281.835} C_VEL
LIN {X 0,Y 296.583,Z 778.293,A -85,B 0,C 180,E1 -16284.418,E2 -16284.418} C_VEL
LIN {X 0,Y 296.504,Z 778.989,A -85,B 0,C 180,E1 -16285.922,E2 -16285.922} C_VEL
LIN {X 0,Y 296.55,Z 779.132,A -85,B 0,C 180,E1 -16287.283,E2 -16287.283} C_VEL
LIN {X 0,Y 296.538,Z 778.846,A -85,B 0,C 180,E1 -16288.642,E2 -16288.642} C_VEL
LIN {X 0,Y 296.509,Z 779.828,A -85,B 0,C 180,E1 -16291.358,E2 -16291.358} C_VEL
LIN {X 0,Y 296.532,Z 780.035,A -85,B 0,C 180,E1 -16292.717,E2 -16292.717} C_VEL
LIN {X 0,Y 296.546,Z 779.306,A -85,B 0,C 180,E1 -16295.509,E2 -16295.509} C_VEL
LIN {X 0,Y 296.867,Z 777.174,A -85,B 0,C 180,E1 -16298.166,E2 -16298.166} C_VEL
LIN {X 0,Y 297.589,Z 773.503,A -85,B 0,C 180,E1 -16300.891,E2 -16300.891} C_VEL
LIN {X 0,Y 298.476,Z 769.769,A -85,B 0,C 180,E1 -16302.926,E2 -16302.926} C_VEL
LIN {X 0,Y 299.708,Z 765.056,A -85,B 0,C 180,E1 -16304.948,E2 -16304.948} C_VEL
LIN {X 0,Y 301.399,Z 758.527,A -85,B 0,C 180,E1 -16307.222,E2 -16307.222} C_VEL
LIN {X 0,Y 303.724,Z 749.976,A -85,B 0,C 180,E1 -16309.604,E2 -16309.604} C_VEL
LIN {X 0,Y 306.119,Z 741.331,A -85,B 0,C 180,E1 -16311.551,E2 -16311.551} C_VEL
LIN {X 0,Y 308.904,Z 730.974,A -85,B 0,C 180,E1 -16313.463,E2 -16313.463} C_VEL
LIN {X 0,Y 311.88,Z 719.554,A -85,B 0,C 180,E1 -16315.172,E2 -16315.172} C_VEL
LIN {X 0,Y 314.612,Z 708.353,A -85,B 0,C 180,E1 -16316.537,E2 -16316.537} C_VEL
LIN {X 0,Y 317.148,Z 696.479,A -85,B 0,C 180,E1 -16317.734,E2 -16317.734} C_VEL
LIN {X 0,Y 319.759,Z 682.622,A -85,B 0,C 180,E1 -16318.827,E2 -16318.827} C_VEL
LIN {X 0,Y 322.244,Z 666.948,A -85,B 0,C 180,E1 -16319.747,E2 -16319.747} C_VEL
LIN {X 0,Y 324.253,Z 648.976,A -85,B 0,C 180,E1 -16320.486,E2 -16320.486} C_VEL
LIN {X 0,Y 330.642,Z 591.432,A -85,B 0,C 180,E1 -16322.592,E2 -16322.592} C_VEL
LIN {X 0,Y 333.332,Z 568.29,A -85,B 0,C 180,E1 -16323.489,E2 -16323.489} C_VEL
LIN {X 0,Y 333.075,Z 566.058,A -85,B 0,C 180,E1 -16323.706,E2 -16323.706} C_VEL
LIN {X 0,Y 329.338,Z 558.398,A -85,B 0,C 180,E1 -16325.343,E2 -16325.343} C_VEL
LIN {X 0,Y 327.097,Z 554.235,A -85,B 0,C 180,E1 -16326.458,E2 -16326.458} C_VEL
LIN {X 0,Y 324.739,Z 550.267,A -85,B 0,C 180,E1 -16327.758,E2 -16327.758} C_VEL
LIN {X 0,Y 321.699,Z 545.672,A -85,B 0,C 180,E1 -16329.764,E2 -16329.764} C_VEL
LIN {X 0,Y 318.601,Z 541.599,A -85,B 0,C 180,E1 -16332.702,E2 -16332.702} C_VEL
LIN {X 0,Y 317.733,Z 540.524,A -85,B 0,C 180,E1 -16334.045,E2 -16334.045} C_VEL
LIN {X 0,Y 316.954,Z 540.047,A -85,B 0,C 180,E1 -16336.577,E2 -16336.577} C_VEL
LIN {X 0,Y 317.397,Z 541.029,A -85,B 0,C 180,E1 -16339.05,E2 -16339.05} C_VEL
LIN {X 0,Y 318.333,Z 542.494,A -85,B 0,C 180,E1 -16340.705,E2 -16340.705} C_VEL
LIN {X 0,Y 321.131,Z 547.636,A -85,B 0,C 180,E1 -16343.69,E2 -16343.69} C_VEL
LIN {X 0,Y 322.304,Z 549.49,A -85,B 0,C 180,E1 -16344.551,E2 -16344.551} C_VEL
LIN {X 0,Y 325.2,Z 555.33,A -85,B 0,C 180,E1 -16346.496,E2 -16346.496} C_VEL
LIN {X 0,Y 327.635,Z 560.574,A -85,B 0,C 180,E1 -16347.863,E2 -16347.863} C_VEL
LIN {X 0,Y 329.005,Z 563.963,A -85,B 0,C 180,E1 -16348.602,E2 -16348.602} C_VEL
LIN {X 0,Y 330.307,Z 575.229,A -85,B 0,C 180,E1 -16349.897,E2 -16349.897} C_VEL
LIN {X 0,Y 331.052,Z 585.515,A -85,B 0,C 180,E1 -16350.851,E2 -16350.851} C_VEL
LIN {X 0,Y 321.803,Z 660.06,A -85,B 0,C 180,E1 -16353.965,E2 -16353.965} C_VEL
LIN {X 0,Y 319.837,Z 672.686,A -85,B 0,C 180,E1 -16354.712,E2 -16354.712} C_VEL
LIN {X 0,Y 317.3,Z 686.743,A -85,B 0,C 180,E1 -16355.81,E2 -16355.81} C_VEL
LIN {X 0,Y 314.866,Z 698.656,A -85,B 0,C 180,E1 -16357.007,E2 -16357.007} C_VEL
LIN {X 0,Y 311.71,Z 711.893,A -85,B 0,C 180,E1 -16358.681,E2 -16358.681} C_VEL
LIN {X 0,Y 308.949,Z 722.691,A -85,B 0,C 180,E1 -16360.395,E2 -16360.395} C_VEL
LIN {X 0,Y 306.213,Z 732.283,A -85,B 0,C 180,E1 -16362.296,E2 -16362.296} C_VEL
LIN {X 0,Y 304.002,Z 740.202,A -85,B 0,C 180,E1 -16364.238,E2 -16364.238} C_VEL
LIN {X 0,Y 302.423,Z 745.631,A -85,B 0,C 180,E1 -16365.877,E2 -16365.877} C_VEL
LIN {X 0,Y 300.63,Z 751.024,A -85,B 0,C 180,E1 -16367.854,E2 -16367.854} C_VEL
LIN {X 0,Y 299.435,Z 755.269,A -85,B 0,C 180,E1 -16369.861,E2 -16369.861} C_VEL
LIN {X 0,Y 298.375,Z 758.466,A -85,B 0,C 180,E1 -16371.875,E2 -16371.875} C_VEL
LIN {X 0,Y 297.757,Z 760.049,A -85,B 0,C 180,E1 -16373.222,E2 -16373.222} C_VEL
LIN {X 0,Y 297.334,Z 761.205,A -85,B 0,C 180,E1 -16374.575,E2 -16374.575} C_VEL
LIN {X 0,Y 297.07,Z 761.914,A -85,B 0,C 180,E1 -16375.93,E2 -16375.93} C_VEL
LIN {X 0,Y 296.834,Z 762.202,A -85,B 0,C 180,E1 -16377.286,E2 -16377.286} C_VEL
LIN {X 0,Y 296.648,Z 762.077,A -85,B 0,C 180,E1 -16378.642,E2 -16378.642} C_VEL
LIN {X 0,Y 296.553,Z 761.536,A -85,B 0,C 180,E1 -16380,E2 -16380} C_VEL
LIN {X 0,Y 296.533,Z 760.542,A -85,B 0,C 180,E1 -16381.358,E2 -16381.358} C_VEL
LIN {X 0,Y 296.583,Z 759.103,A -85,B 0,C 180,E1 -16382.716,E2 -16382.716} C_VEL
LIN {X 0,Y 296.575,Z 756.1,A -85,B 0,C 180,E1 -16384.758,E2 -16384.758} C_VEL
LIN {X 0,Y 296.775,Z 751.988,A -85,B 0,C 180,E1 -16386.8,E2 -16386.8} C_VEL
LIN {X 0,Y 297.136,Z 745.652,A -85,B 0,C 180,E1 -16389.187,E2 -16389.187} C_VEL
LIN {X 0,Y 297.651,Z 738.71,A -85,B 0,C 180,E1 -16391.233,E2 -16391.233} C_VEL
LIN {X 0,Y 298.454,Z 730.093,A -85,B 0,C 180,E1 -16393.273,E2 -16393.273} C_VEL
LIN {X 0,Y 299.218,Z 719.81,A -85,B 0,C 180,E1 -16395.25,E2 -16395.25} C_VEL
LIN {X 0,Y 300.367,Z 708.38,A -85,B 0,C 180,E1 -16397.006,E2 -16397.006} C_VEL
LIN {X 0,Y 301.472,Z 696.166,A -85,B 0,C 180,E1 -16398.52,E2 -16398.52} C_VEL
LIN {X 0,Y 302.442,Z 684.283,A -85,B 0,C 180,E1 -16399.691,E2 -16399.691} C_VEL
LIN {X 0,Y 303.31,Z 671.328,A -85,B 0,C 180,E1 -16400.693,E2 -16400.693} C_VEL
LIN {X 0,Y 304.16,Z 657.438,A -85,B 0,C 180,E1 -16401.475,E2 -16401.475} C_VEL
LIN {X 0,Y 305.192,Z 633.134,A -85,B 0,C 180,E1 -16402.376,E2 -16402.376} C_VEL
LIN {X 0,Y 307.542,Z 575.725,A -85,B 0,C 180,E1 -16404.369,E2 -16404.369} C_VEL
LIN {X 0,Y 303.488,Z 542.01,A -85,B 0,C 180,E1 -16405.844,E2 -16405.844} C_VEL
LIN {X 0,Y 303.245,Z 538.749,A -85,B 0,C 180,E1 -16406.024,E2 -16406.024} C_VEL
LIN {X 0,Y 304.722,Z 527.448,A -85,B 0,C 180,E1 -16408.786,E2 -16408.786} C_VEL
LIN {X 0,Y 301.943,Z 514.34,A -85,B 0,C 180,E1 -16412.367,E2 -16412.367} C_VEL
LIN {X 0,Y 299.184,Z 501.713,A -85,B 0,C 180,E1 -16415.963,E2 -16415.963} C_VEL
LIN {X 0,Y 298.468,Z 498.43,A -85,B 0,C 180,E1 -16416.963,E2 -16416.963} C_VEL
LIN {X 0,Y 298.414,Z 498.437,A -85,B 0,C 180,E1 -16421.257,E2 -16421.257} C_VEL
LIN {X 0,Y 298.355,Z 498.444,A -85,B 0,C 180,E1 -16425.035,E2 -16425.035} C_VEL
LIN {X 0,Y 298.385,Z 498.439,A -85,B 0,C 180,E1 -16428.738,E2 -16428.738} C_VEL
LIN {X 0,Y 298.415,Z 498.436,A -85,B 0,C 180,E1 -16432.242,E2 -16432.242} C_VEL
LIN {X 0,Y 298.41,Z 498.44,A -85,B 0,C 180,E1 -16435.581,E2 -16435.581} C_VEL
LIN {X 0,Y 298.397,Z 498.438,A -85,B 0,C 180,E1 -16438.791,E2 -16438.791} C_VEL
LIN {X 0,Y 298.465,Z 498.431,A -85,B 0,C 180,E1 -16441.904,E2 -16441.904} C_VEL
LIN {X 0,Y 298.487,Z 498.426,A -85,B 0,C 180,E1 -16444.924,E2 -16444.924} C_VEL
LIN {X 0,Y 298.453,Z 498.434,A -85,B 0,C 180,E1 -16449.315,E2 -16449.315} C_VEL
LIN {X 0,Y 298.539,Z 498.419,A -85,B 0,C 180,E1 -16452.179,E2 -16452.179} C_VEL
LIN {X 0,Y 298.595,Z 498.414,A -85,B 0,C 180,E1 -16454.995,E2 -16454.995} C_VEL
LIN {X 0,Y 298.595,Z 498.415,A -85,B 0,C 180,E1 -16459.147,E2 -16459.147} C_VEL
LIN {X 0,Y 298.76,Z 498.394,A -85,B 0,C 180,E1 -16461.886,E2 -16461.886} C_VEL
LIN {X 0,Y 298.662,Z 498.404,A -85,B 0,C 180,E1 -16464.599,E2 -16464.599} C_VEL
LIN {X 0,Y 298.928,Z 498.371,A -85,B 0,C 180,E1 -16468.653,E2 -16468.653} C_VEL
LIN {X 0,Y 298.926,Z 498.376,A -85,B 0,C 180,E1 -16471.347,E2 -16471.347} C_VEL
LIN {X 0,Y 298.799,Z 498.388,A -85,B 0,C 180,E1 -16476.754,E2 -16476.754} C_VEL
LIN {X 0,Y 298.682,Z 498.407,A -85,B 0,C 180,E1 -16479.48,E2 -16479.48} C_VEL
LIN {X 0,Y 298.554,Z 498.421,A -85,B 0,C 180,E1 -16483.615,E2 -16483.615} C_VEL
LIN {X 0,Y 298.55,Z 498.418,A -85,B 0,C 180,E1 -16486.409,E2 -16486.409} C_VEL
LIN {X 0,Y 298.513,Z 498.426,A -85,B 0,C 180,E1 -16489.655,E2 -16489.655} C_VEL
LIN {X 0,Y 298.459,Z 498.432,A -85,B 0,C 180,E1 -16493.598,E2 -16493.598} C_VEL
LIN {X 0,Y 298.486,Z 498.426,A -85,B 0,C 180,E1 -16496.575,E2 -16496.575} C_VEL
LIN {X 0,Y 298.417,Z 498.438,A -85,B 0,C 180,E1 -16499.641,E2 -16499.641} C_VEL
LIN {X 0,Y 298.396,Z 498.438,A -85,B 0,C 180,E1 -16502.8,E2 -16502.8} C_VEL
LIN {X 0,Y 298.466,Z 498.43,A -85,B 0,C 180,E1 -16506.812,E2 -16506.812} C_VEL
LIN {X 0,Y 298.389,Z 498.441,A -85,B 0,C 180,E1 -16511.088,E2 -16511.088} C_VEL
LIN {X 0,Y 298.389,Z 498.441,A -85,B 0,C 180,E1 -16515.042,E2 -16515.042} C_VEL
LIN {X 0,Y 298.389,Z 498.44,A -85,B 0,C 180,E1 -16518.912,E2 -16518.912} C_VEL
LIN {X 0,Y 298.447,Z 498.436,A -85,B 0,C 180,E1 -16523.192,E2 -16523.192} C_VEL
LIN {X 0,Y 298.444,Z 498.537,A -85,B 0,C 180,E1 -16525.765,E2 -16525.765} C_VEL
LIN {X 0,Y 302.073,Z 514.185,A -85,B 0,C 180,E1 -16529.213,E2 -16529.213} C_VEL
LIN {X 0,Y 304.733,Z 526.676,A -85,B 0,C 180,E1 -16531.887,E2 -16531.887} C_VEL
LIN {X 0,Y 303.576,Z 542.048,A -85,B 0,C 180,E1 -16534.88,E2 -16534.88} C_VEL
LIN {X 0,Y 302.981,Z 549.388,A -85,B 0,C 180,E1 -16536.3,E2 -16536.3} C_VEL
LIN {X 0,Y 305.486,Z 572.218,A -85,B 0,C 180,E1 -16537.229,E2 -16537.229} C_VEL
LIN {X 0,Y 306.131,Z 579.488,A -85,B 0,C 180,E1 -16537.514,E2 -16537.514} C_VEL
LIN {X 0,Y 305.977,Z 583.656,A -85,B 0,C 180,E1 -16537.651,E2 -16537.651} C_VEL
LIN {X 0,Y 305.054,Z 589.436,A -85,B 0,C 180,E1 -16537.814,E2 -16537.814} C_VEL
LIN {X 0,Y 298.705,Z 608.105,A -85,B 0,C 180,E1 -16538.242,E2 -16538.242} C_VEL
LIN {X 0,Y 297.871,Z 613.874,A -85,B 0,C 180,E1 -16538.427,E2 -16538.427} C_VEL
LIN {X 0,Y 296.242,Z 660.915,A -85,B 0,C 180,E1 -16540.106,E2 -16540.106} C_VEL
LIN {X 0,Y 295.582,Z 674.395,A -85,B 0,C 180,E1 -16540.827,E2 -16540.827} C_VEL
LIN {X 0,Y 294.667,Z 688.96,A -85,B 0,C 180,E1 -16541.937,E2 -16541.937} C_VEL
LIN {X 0,Y 293.727,Z 700.985,A -85,B 0,C 180,E1 -16543.153,E2 -16543.153} C_VEL
LIN {X 0,Y 292.813,Z 713.045,A -85,B 0,C 180,E1 -16544.691,E2 -16544.691} C_VEL
LIN {X 0,Y 291.883,Z 723.847,A -85,B 0,C 180,E1 -16546.422,E2 -16546.422} C_VEL
LIN {X 0,Y 291.082,Z 732.727,A -85,B 0,C 180,E1 -16548.157,E2 -16548.157} C_VEL
LIN {X 0,Y 290.385,Z 741.35,A -85,B 0,C 180,E1 -16550.246,E2 -16550.246} C_VEL
LIN {X 0,Y 289.923,Z 748.265,A -85,B 0,C 180,E1 -16552.338,E2 -16552.338} C_VEL
LIN {X 0,Y 289.645,Z 753.753,A -85,B 0,C 180,E1 -16554.43,E2 -16554.43} C_VEL
LIN {X 0,Y 289.552,Z 757.968,A -85,B 0,C 180,E1 -16556.521,E2 -16556.521} C_VEL
LIN {X 0,Y 289.423,Z 761.052,A -85,B 0,C 180,E1 -16558.609,E2 -16558.609} C_VEL
LIN {X 0,Y 289.434,Z 762.517,A -85,B 0,C 180,E1 -16560,E2 -16560} C_VEL
LIN {X 0,Y 289.473,Z 763.563,A -85,B 0,C 180,E1 -16561.391,E2 -16561.391} C_VEL
LIN {X 0,Y 289.588,Z 764.147,A -85,B 0,C 180,E1 -16562.782,E2 -16562.782} C_VEL
LIN {X 0,Y 289.766,Z 764.283,A -85,B 0,C 180,E1 -16564.173,E2 -16564.173} C_VEL
LIN {X 0,Y 290.069,Z 764.009,A -85,B 0,C 180,E1 -16565.562,E2 -16565.562} C_VEL
LIN {X 0,Y 290.637,Z 762.884,A -85,B 0,C 180,E1 -16567.502,E2 -16567.502} C_VEL
LIN {X 0,Y 291.405,Z 760.573,A -85,B 0,C 180,E1 -16569.719,E2 -16569.719} C_VEL
LIN {X 0,Y 292.545,Z 757.353,A -85,B 0,C 180,E1 -16571.783,E2 -16571.783} C_VEL
LIN {X 0,Y 293.88,Z 753.08,A -85,B 0,C 180,E1 -16573.836,E2 -16573.836} C_VEL
LIN {X 0,Y 296.019,Z 746.512,A -85,B 0,C 180,E1 -16576.199,E2 -16576.199} C_VEL
LIN {X 0,Y 298.662,Z 738.091,A -85,B 0,C 180,E1 -16578.523,E2 -16578.523} C_VEL
LIN {X 0,Y 301.317,Z 728.987,A -85,B 0,C 180,E1 -16580.479,E2 -16580.479} C_VEL
LIN {X 0,Y 303.814,Z 719.537,A -85,B 0,C 180,E1 -16582.116,E2 -16582.116} C_VEL
LIN {X 0,Y 306.679,Z 707.342,A -85,B 0,C 180,E1 -16583.822,E2 -16583.822} C_VEL
LIN {X 0,Y 309.168,Z 695.987,A -85,B 0,C 180,E1 -16585.048,E2 -16585.048} C_VEL
LIN {X 0,Y 311.59,Z 682.547,A -85,B 0,C 180,E1 -16586.183,E2 -16586.183} C_VEL
LIN {X 0,Y 313.513,Z 669.748,A -85,B 0,C 180,E1 -16586.997,E2 -16586.997} C_VEL
LIN {X 0,Y 315.151,Z 655.434,A -85,B 0,C 180,E1 -16587.654,E2 -16587.654} C_VEL
LIN {X 0,Y 322.826,Z 588.936,A -85,B 0,C 180,E1 -16590.334,E2 -16590.334} C_VEL
LIN {X 0,Y 321.846,Z 578.296,A -85,B 0,C 180,E1 -16591.365,E2 -16591.365} C_VEL
LIN {X 0,Y 320.291,Z 565.64,A -85,B 0,C 180,E1 -16592.848,E2 -16592.848} C_VEL
LIN {X 0,Y 319.589,Z 561.659,A -85,B 0,C 180,E1 -16593.422,E2 -16593.422} C_VEL
LIN {X 0,Y 317.578,Z 556.682,A -85,B 0,C 180,E1 -16594.606,E2 -16594.606} C_VEL
LIN {X 0,Y 316.475,Z 553.652,A -85,B 0,C 180,E1 -16595.45,E2 -16595.45} C_VEL
LIN {X 0,Y 315.962,Z 548.674,A -85,B 0,C 180,E1 -16597.805,E2 -16597.805} C_VEL
LIN {X 0,Y 315.482,Z 544.781,A -85,B 0,C 180,E1 -16600.243,E2 -16600.243} C_VEL
LIN {X 0,Y 315.181,Z 542.315,A -85,B 0,C 180,E1 -16602.621,E2 -16602.621} C_VEL
LIN {X 0,Y 315.231,Z 541.208,A -85,B 0,C 180,E1 -16604.485,E2 -16604.485} C_VEL
LIN {X 0,Y 315.829,Z 540.857,A -85,B 0,C 180,E1 -16607.251,E2 -16607.251} C_VEL
LIN {X 0,Y 317.193,Z 542.15,A -85,B 0,C 180,E1 -16610.018,E2 -16610.018} C_VEL
LIN {X 0,Y 319.227,Z 544.595,A -85,B 0,C 180,E1 -16612.426,E2 -16612.426} C_VEL
LIN {X 0,Y 320.878,Z 547.738,A -85,B 0,C 180,E1 -16614.134,E2 -16614.134} C_VEL
LIN {X 0,Y 321.548,Z 555.584,A -85,B 0,C 180,E1 -16616.156,E2 -16616.156} C_VEL
LIN {X 0,Y 322.001,Z 558.563,A -85,B 0,C 180,E1 -16616.791,E2 -16616.791} C_VEL
LIN {X 0,Y 322.043,Z 569.404,A -85,B 0,C 180,E1 -16617.689,E2 -16617.689} C_VEL
LIN {X 0,Y 311.746,Z 655.982,A -85,B 0,C 180,E1 -16621.422,E2 -16621.422} C_VEL
LIN {X 0,Y 309.197,Z 680.233,A -85,B 0,C 180,E1 -16622.54,E2 -16622.54} C_VEL
LIN {X 0,Y 307.309,Z 693.753,A -85,B 0,C 180,E1 -16623.414,E2 -16623.414} C_VEL
LIN {X 0,Y 305.363,Z 705.817,A -85,B 0,C 180,E1 -16624.463,E2 -16624.463} C_VEL
LIN {X 0,Y 303.254,Z 717.349,A -85,B 0,C 180,E1 -16625.71,E2 -16625.71} C_VEL
LIN {X 0,Y 300.727,Z 729.268,A -85,B 0,C 180,E1 -16627.319,E2 -16627.319} C_VEL
LIN {X 0,Y 298.455,Z 739.127,A -85,B 0,C 180,E1 -16628.955,E2 -16628.955} C_VEL
LIN {X 0,Y 296.176,Z 748.806,A -85,B 0,C 180,E1 -16630.957,E2 -16630.957} C_VEL
LIN {X 0,Y 294.221,Z 756.787,A -85,B 0,C 180,E1 -16632.985,E2 -16632.985} C_VEL
LIN {X 0,Y 292.498,Z 764.195,A -85,B 0,C 180,E1 -16635.387,E2 -16635.387} C_VEL
LIN {X 0,Y 291.289,Z 769.236,A -85,B 0,C 180,E1 -16637.459,E2 -16637.459} C_VEL
LIN {X 0,Y 290.407,Z 773.151,A -85,B 0,C 180,E1 -16639.543,E2 -16639.543} C_VEL
LIN {X 0,Y 289.867,Z 776.015,A -85,B 0,C 180,E1 -16641.635,E2 -16641.635} C_VEL
LIN {X 0,Y 289.633,Z 777.402,A -85,B 0,C 180,E1 -16643.031,E2 -16643.031} C_VEL
LIN {X 0,Y 289.5,Z 778.342,A -85,B 0,C 180,E1 -16644.46,E2 -16644.46} C_VEL
LIN {X 0,Y 289.412,Z 778.81,A -85,B 0,C 180,E1 -16645.822,E2 -16645.822} C_VEL
LIN {X 0,Y 289.473,Z 778.878,A -85,B 0,C 180,E1 -16647.217,E2 -16647.217} C_VEL
LIN {X 0,Y 289.469,Z 778.34,A -85,B 0,C 180,E1 -16649.305,E2 -16649.305} C_VEL
LIN {X 0,Y 289.429,Z 779.462,A -85,B 0,C 180,E1 -16651.392,E2 -16651.392} C_VEL
LIN {X 0,Y 289.456,Z 779.742,A -85,B 0,C 180,E1 -16652.783,E2 -16652.783} C_VEL
LIN {X 0,Y 289.476,Z 779.19,A -85,B 0,C 180,E1 -16655.573,E2 -16655.573} C_VEL
LIN {X 0,Y 289.825,Z 777.196,A -85,B 0,C 180,E1 -16658.366,E2 -16658.366} C_VEL
LIN {X 0,Y 290.607,Z 773.741,A -85,B 0,C 180,E1 -16661.156,E2 -16661.156} C_VEL
LIN {X 0,Y 291.538,Z 770.113,A -85,B 0,C 180,E1 -16663.239,E2 -16663.239} C_VEL
LIN {X 0,Y 292.842,Z 765.584,A -85,B 0,C 180,E1 -16665.307,E2 -16665.307} C_VEL
LIN {X 0,Y 294.654,Z 759.331,A -85,B 0,C 180,E1 -16667.606,E2 -16667.606} C_VEL
LIN {X 0,Y 297.123,Z 750.993,A -85,B 0,C 180,E1 -16670.058,E2 -16670.058} C_VEL
LIN {X 0,Y 299.638,Z 742.654,A -85,B 0,C 180,E1 -16672.042,E2 -16672.042} C_VEL
LIN {X 0,Y 302.58,Z 732.717,A -85,B 0,C 180,E1 -16673.984,E2 -16673.984} C_VEL
LIN {X 0,Y 305.996,Z 720.631,A -85,B 0,C 180,E1 -16675.874,E2 -16675.874} C_VEL
LIN {X 0,Y 309.179,Z 708.44,A -85,B 0,C 180,E1 -16677.407,E2 -16677.407} C_VEL
LIN {X 0,Y 311.857,Z 696.755,A -85,B 0,C 180,E1 -16678.613,E2 -16678.613} C_VEL
LIN {X 0,Y 314.643,Z 683.246,A -85,B 0,C 180,E1 -16679.709,E2 -16679.709} C_VEL
LIN {X 0,Y 317.356,Z 667.356,A -85,B 0,C 180,E1 -16680.667,E2 -16680.667} C_VEL
LIN {X 0,Y 319.4,Z 651.035,A -85,B 0,C 180,E1 -16681.368,E2 -16681.368} C_VEL
LIN {X 0,Y 327.548,Z 583.603,A -85,B 0,C 180,E1 -16683.909,E2 -16683.909} C_VEL
LIN {X 0,Y 329.185,Z 570.446,A -85,B 0,C 180,E1 -16684.448,E2 -16684.448} C_VEL
LIN {X 0,Y 326.101,Z 563.759,A -85,B 0,C 180,E1 -16685.944,E2 -16685.944} C_VEL
LIN {X 0,Y 324.161,Z 560.036,A -85,B 0,C 180,E1 -16686.961,E2 -16686.961} C_VEL
LIN {X 0,Y 322.061,Z 556.341,A -85,B 0,C 180,E1 -16688.224,E2 -16688.224} C_VEL
LIN {X 0,Y 319.396,Z 552.147,A -85,B 0,C 180,E1 -16690.111,E2 -16690.111} C_VEL
LIN {X 0,Y 316.699,Z 548.336,A -85,B 0,C 180,E1 -16692.919,E2 -16692.919} C_VEL
LIN {X 0,Y 315.964,Z 547.353,A -85,B 0,C 180,E1 -16694.168,E2 -16694.168} C_VEL
LIN {X 0,Y 315.274,Z 546.958,A -85,B 0,C 180,E1 -16696.287,E2 -16696.287} C_VEL
LIN {X 0,Y 315.517,Z 547.679,A -85,B 0,C 180,E1 -16698.696,E2 -16698.696} C_VEL
LIN {X 0,Y 316.437,Z 549.296,A -85,B 0,C 180,E1 -16700.551,E2 -16700.551} C_VEL
LIN {X 0,Y 319.182,Z 554.56,A -85,B 0,C 180,E1 -16703.639,E2 -16703.639} C_VEL
LIN {X 0,Y 320.317,Z 556.97,A -85,B 0,C 180,E1 -16704.565,E2 -16704.565} C_VEL
LIN {X 0,Y 322.451,Z 561.424,A -85,B 0,C 180,E1 -16706.06,E2 -16706.06} C_VEL
LIN {X 0,Y 324.701,Z 566.692,A -85,B 0,C 180,E1 -16707.452,E2 -16707.452} C_VEL
LIN {X 0,Y 325.433,Z 568.921,A -85,B 0,C 180,E1 -16707.911,E2 -16707.911} C_VEL
LIN {X 0,Y 326.342,Z 578.672,A -85,B 0,C 180,E1 -16709.06,E2 -16709.06} C_VEL
LIN {X 0,Y 326.798,Z 587.167,A -85,B 0,C 180,E1 -16709.891,E2 -16709.891} C_VEL
LIN {X 0,Y 316.944,Z 660.969,A -85,B 0,C 180,E1 -16713.052,E2 -16713.052} C_VEL
LIN {X 0,Y 314.793,Z 673.857,A -85,B 0,C 180,E1 -16713.836,E2 -16713.836} C_VEL
LIN {X 0,Y 311.926,Z 688.257,A -85,B 0,C 180,E1 -16715.01,E2 -16715.01} C_VEL
LIN {X 0,Y 309.03,Z 701.079,A -85,B 0,C 180,E1 -16716.37,E2 -16716.37} C_VEL
LIN {X 0,Y 306.017,Z 712.825,A -85,B 0,C 180,E1 -16717.91,E2 -16717.91} C_VEL
LIN {X 0,Y 303.052,Z 723.34,A -85,B 0,C 180,E1 -16719.643,E2 -16719.643} C_VEL
LIN {X 0,Y 300.138,Z 732.901,A -85,B 0,C 180,E1 -16721.572,E2 -16721.572} C_VEL
LIN {X 0,Y 297.717,Z 740.69,A -85,B 0,C 180,E1 -16723.544,E2 -16723.544} C_VEL
LIN {X 0,Y 295.68,Z 747.059,A -85,B 0,C 180,E1 -16725.548,E2 -16725.548} C_VEL
LIN {X 0,Y 293.807,Z 752.235,A -85,B 0,C 180,E1 -16727.568,E2 -16727.568} C_VEL
LIN {X 0,Y 292.52,Z 756.228,A -85,B 0,C 180,E1 -16729.619,E2 -16729.619} C_VEL
LIN {X 0,Y 291.395,Z 759.222,A -85,B 0,C 180,E1 -16731.679,E2 -16731.679} C_VEL
LIN {X 0,Y 290.754,Z 760.697,A -85,B 0,C 180,E1 -16733.058,E2 -16733.058} C_VEL
LIN {X 0,Y 290.298,Z 761.704,A -85,B 0,C 180,E1 -16734.443,E2 -16734.443} C_VEL
LIN {X 0,Y 290.007,Z 762.299,A -85,B 0,C 180,E1 -16735.831,E2 -16735.831} C_VEL
LIN {X 0,Y 289.759,Z 762.493,A -85,B 0,C 180,E1 -16737.219,E2 -16737.219} C_VEL
LIN {X 0,Y 289.566,Z 762.277,A -85,B 0,C 180,E1 -16738.609,E2 -16738.609} C_VEL
LIN {X 0,Y 289.469,Z 761.598,A -85,B 0,C 180,E1 -16740,E2 -16740} C_VEL
LIN {X 0,Y 289.453,Z 760.489,A -85,B 0,C 180,E1 -16741.391,E2 -16741.391} C_VEL
LIN {X 0,Y 289.486,Z 758.957,A -85,B 0,C 180,E1 -16742.783,E2 -16742.783} C_VEL
LIN {X 0,Y 289.499,Z 755.486,A -85,B 0,C 180,E1 -16745.045,E2 -16745.045} C_VEL
LIN {X 0,Y 289.753,Z 750.768,A -85,B 0,C 180,E1 -16747.27,E2 -16747.27} C_VEL
LIN {X 0,Y 290.097,Z 744.947,A -85,B 0,C 180,E1 -16749.412,E2 -16749.412} C_VEL
LIN {X 0,Y 290.626,Z 737.737,A -85,B 0,C 180,E1 -16751.508,E2 -16751.508} C_VEL
LIN {X 0,Y 291.482,Z 728.863,A -85,B 0,C 180,E1 -16753.597,E2 -16753.597} C_VEL
LIN {X 0,Y 292.152,Z 719.79,A -85,B 0,C 180,E1 -16755.344,E2 -16755.344} C_VEL
LIN {X 0,Y 293.279,Z 708.804,A -85,B 0,C 180,E1 -16757.071,E2 -16757.071} C_VEL
LIN {X 0,Y 294.391,Z 696.652,A -85,B 0,C 180,E1 -16758.621,E2 -16758.621} C_VEL
LIN {X 0,Y 295.521,Z 682.936,A -85,B 0,C 180,E1 -16759.99,E2 -16759.99} C_VEL
LIN {X 0,Y 296.392,Z 669.55,A -85,B 0,C 180,E1 -16761.017,E2 -16761.017} C_VEL
LIN {X 0,Y 297.237,Z 655.082,A -85,B 0,C 180,E1 -16761.818,E2 -16761.818} C_VEL
LIN {X 0,Y 300.657,Z 576.329,A -85,B 0,C 180,E1 -16764.696,E2 -16764.696} C_VEL
LIN {X 0,Y 296.86,Z 544.867,A -85,B 0,C 180,E1 -16766.101,E2 -16766.101} C_VEL
LIN {X 0,Y 296.374,Z 538.669,A -85,B 0,C 180,E1 -16766.41,E2 -16766.41} C_VEL
LIN {X 0,Y 297.637,Z 529.738,A -85,B 0,C 180,E1 -16768.64,E2 -16768.64} C_VEL
LIN {X 0,Y 297.451,Z 527.076,A -85,B 0,C 180,E1 -16769.342,E2 -16769.342} C_VEL
LIN {X 0,Y 294.41,Z 512.866,A -85,B 0,C 180,E1 -16773.331,E2 -16773.331} C_VEL
LIN {X 0,Y 291.621,Z 500.23,A -85,B 0,C 180,E1 -16777.049,E2 -16777.049} C_VEL
LIN {X 0,Y 291.409,Z 499.309,A -85,B 0,C 180,E1 -16777.354,E2 -16777.354} C_VEL
LIN {X 0,Y 291.352,Z 499.314,A -85,B 0,C 180,E1 -16780.639,E2 -16780.639} C_VEL
LIN {X 0,Y 291.291,Z 499.323,A -85,B 0,C 180,E1 -16784.402,E2 -16784.402} C_VEL
LIN {X 0,Y 291.328,Z 499.319,A -85,B 0,C 180,E1 -16788.404,E2 -16788.404} C_VEL
LIN {X 0,Y 291.355,Z 499.317,A -85,B 0,C 180,E1 -16791.158,E2 -16791.158} C_VEL
LIN {X 0,Y 291.362,Z 499.313,A -85,B 0,C 180,E1 -16794.626,E2 -16794.626} C_VEL
LIN {X 0,Y 291.374,Z 499.314,A -85,B 0,C 180,E1 -16797.951,E2 -16797.951} C_VEL
LIN {X 0,Y 291.384,Z 499.313,A -85,B 0,C 180,E1 -16801.158,E2 -16801.158} C_VEL
LIN {X 0,Y 291.418,Z 499.306,A -85,B 0,C 180,E1 -16804.272,E2 -16804.272} C_VEL
LIN {X 0,Y 291.383,Z 499.314,A -85,B 0,C 180,E1 -16807.299,E2 -16807.299} C_VEL
LIN {X 0,Y 291.46,Z 499.302,A -85,B 0,C 180,E1 -16810.27,E2 -16810.27} C_VEL
LIN {X 0,Y 291.556,Z 499.289,A -85,B 0,C 180,E1 -16814.624,E2 -16814.624} C_VEL
LIN {X 0,Y 291.539,Z 499.293,A -85,B 0,C 180,E1 -16818.881,E2 -16818.881} C_VEL
LIN {X 0,Y 291.711,Z 499.273,A -85,B 0,C 180,E1 -16821.688,E2 -16821.688} C_VEL
LIN {X 0,Y 291.633,Z 499.28,A -85,B 0,C 180,E1 -16824.468,E2 -16824.468} C_VEL
LIN {X 0,Y 291.894,Z 499.247,A -85,B 0,C 180,E1 -16828.62,E2 -16828.62} C_VEL
LIN {X 0,Y 291.892,Z 499.252,A -85,B 0,C 180,E1 -16831.38,E2 -16831.38} C_VEL
LIN {X 0,Y 291.747,Z 499.267,A -85,B 0,C 180,E1 -16836.918,E2 -16836.918} C_VEL
LIN {X 0,Y 291.63,Z 499.283,A -85,B 0,C 180,E1 -16839.712,E2 -16839.712} C_VEL
LIN {X 0,Y 291.523,Z 499.295,A -85,B 0,C 180,E1 -16843.95,E2 -16843.95} C_VEL
LIN {X 0,Y 291.488,Z 499.298,A -85,B 0,C 180,E1 -16846.818,E2 -16846.818} C_VEL
LIN {X 0,Y 291.452,Z 499.304,A -85,B 0,C 180,E1 -16849.875,E2 -16849.875} C_VEL
LIN {X 0,Y 291.4,Z 499.308,A -85,B 0,C 180,E1 -16854.205,E2 -16854.205} C_VEL
LIN {X 0,Y 291.42,Z 499.311,A -85,B 0,C 180,E1 -16857.272,E2 -16857.272} C_VEL
LIN {X 0,Y 291.335,Z 499.317,A -85,B 0,C 180,E1 -16860.437,E2 -16860.437} C_VEL
LIN {X 0,Y 291.345,Z 499.317,A -85,B 0,C 180,E1 -16863.698,E2 -16863.698} C_VEL
LIN {X 0,Y 291.396,Z 499.314,A -85,B 0,C 180,E1 -16867.259,E2 -16867.259} C_VEL
LIN {X 0,Y 291.336,Z 499.317,A -85,B 0,C 180,E1 -16870.642,E2 -16870.642} C_VEL
LIN {X 0,Y 291.315,Z 499.319,A -85,B 0,C 180,E1 -16874.397,E2 -16874.397} C_VEL
LIN {X 0,Y 291.328,Z 499.318,A -85,B 0,C 180,E1 -16878.404,E2 -16878.404} C_VEL
LIN {X 0,Y 291.354,Z 499.319,A -85,B 0,C 180,E1 -16881.159,E2 -16881.159} C_VEL
LIN {X 0,Y 291.363,Z 499.315,A -85,B 0,C 180,E1 -16884.626,E2 -16884.626} C_VEL
LIN {X 0,Y 291.405,Z 499.509,A -85,B 0,C 180,E1 -16885.431,E2 -16885.431} C_VEL
LIN {X 0,Y 295.119,Z 515.503,A -85,B 0,C 180,E1 -16889.016,E2 -16889.016} C_VEL
LIN {X 0,Y 297.791,Z 528.487,A -85,B 0,C 180,E1 -16891.835,E2 -16891.835} C_VEL
LIN {X 0,Y 296.079,Z 549.477,A -85,B 0,C 180,E1 -16895.969,E2 -16895.969} C_VEL
LIN {X 0,Y 298.287,Z 571.024,A -85,B 0,C 180,E1 -16896.871,E2 -16896.871} C_VEL
LIN {X 0,Y 299.209,Z 579.826,A -85,B 0,C 180,E1 -16897.236,E2 -16897.236} C_VEL
LIN {X 0,Y 297.871,Z 613.874,A -85,B 0,C 180,E1 -16898.427,E2 -16898.427} C_VEL
LIN {X 0,Y 297.019,Z 619.645,A -85,B 0,C 180,E1 -16898.609,E2 -16898.609} C_VEL
LIN {X 0,Y 290.702,Z 638.307,A -85,B 0,C 180,E1 -16899.083,E2 -16899.083} C_VEL
LIN {X 0,Y 289.889,Z 644.079,A -85,B 0,C 180,E1 -16899.275,E2 -16899.275} C_VEL
LIN {X 0,Y 289.058,Z 664.82,A -85,B 0,C 180,E1 -16900.099,E2 -16900.099} C_VEL
LIN {X 0,Y 288.284,Z 678.987,A -85,B 0,C 180,E1 -16900.97,E2 -16900.97} C_VEL
LIN {X 0,Y 287.485,Z 691.448,A -85,B 0,C 180,E1 -16902.023,E2 -16902.023} C_VEL
LIN {X 0,Y 286.415,Z 703.424,A -85,B 0,C 180,E1 -16903.315,E2 -16903.315} C_VEL
LIN {X 0,Y 285.673,Z 713.442,A -85,B 0,C 180,E1 -16904.665,E2 -16904.665} C_VEL
LIN {X 0,Y 284.754,Z 724.179,A -85,B 0,C 180,E1 -16906.44,E2 -16906.44} C_VEL
LIN {X 0,Y 283.977,Z 733.013,A -85,B 0,C 180,E1 -16908.219,E2 -16908.219} C_VEL
LIN {X 0,Y 283.282,Z 741.597,A -85,B 0,C 180,E1 -16910.36,E2 -16910.36} C_VEL
LIN {X 0,Y 282.817,Z 748.525,A -85,B 0,C 180,E1 -16912.504,E2 -16912.504} C_VEL
LIN {X 0,Y 282.512,Z 754.351,A -85,B 0,C 180,E1 -16914.807,E2 -16914.807} C_VEL
LIN {X 0,Y 282.456,Z 758.804,A -85,B 0,C 180,E1 -16917.148,E2 -16917.148} C_VEL
LIN {X 0,Y 282.348,Z 760.88,A -85,B 0,C 180,E1 -16918.574,E2 -16918.574} C_VEL
LIN {X 0,Y 282.354,Z 762.448,A -85,B 0,C 180,E1 -16920,E2 -16920} C_VEL
LIN {X 0,Y 282.396,Z 763.568,A -85,B 0,C 180,E1 -16921.426,E2 -16921.426} C_VEL
LIN {X 0,Y 282.52,Z 764.28,A -85,B 0,C 180,E1 -16922.852,E2 -16922.852} C_VEL
LIN {X 0,Y 282.695,Z 764.545,A -85,B 0,C 180,E1 -16924.277,E2 -16924.277} C_VEL
LIN {X 0,Y 283.021,Z 764.357,A -85,B 0,C 180,E1 -16925.701,E2 -16925.701} C_VEL
LIN {X 0,Y 283.602,Z 763.475,A -85,B 0,C 180,E1 -16927.585,E2 -16927.585} C_VEL
LIN {X 0,Y 284.439,Z 761.289,A -85,B 0,C 180,E1 -16929.96,E2 -16929.96} C_VEL
LIN {X 0,Y 285.664,Z 758.27,A -85,B 0,C 180,E1 -16932.071,E2 -16932.071} C_VEL
LIN {X 0,Y 287.08,Z 754.181,A -85,B 0,C 180,E1 -16934.171,E2 -16934.171} C_VEL
LIN {X 0,Y 289.349,Z 747.96,A -85,B 0,C 180,E1 -16936.583,E2 -16936.583} C_VEL
LIN {X 0,Y 291.705,Z 741.156,A -85,B 0,C 180,E1 -16938.616,E2 -16938.616} C_VEL
LIN {X 0,Y 294.425,Z 732.723,A -85,B 0,C 180,E1 -16940.615,E2 -16940.615} C_VEL
LIN {X 0,Y 296.974,Z 724.31,A -85,B 0,C 180,E1 -16942.25,E2 -16942.25} C_VEL
LIN {X 0,Y 299.781,Z 713.878,A -85,B 0,C 180,E1 -16943.892,E2 -16943.892} C_VEL
LIN {X 0,Y 302.459,Z 702.911,A -85,B 0,C 180,E1 -16945.275,E2 -16945.275} C_VEL
LIN {X 0,Y 305.168,Z 690.59,A -85,B 0,C 180,E1 -16946.501,E2 -16946.501} C_VEL
LIN {X 0,Y 307.623,Z 676.782,A -85,B 0,C 180,E1 -16947.557,E2 -16947.557} C_VEL
LIN {X 0,Y 309.712,Z 661.795,A -85,B 0,C 180,E1 -16948.367,E2 -16948.367} C_VEL
LIN {X 0,Y 318.534,Z 590.692,A -85,B 0,C 180,E1 -16951.313,E2 -16951.313} C_VEL
LIN {X 0,Y 317.707,Z 579.764,A -85,B 0,C 180,E1 -16952.435,E2 -16952.435} C_VEL
LIN {X 0,Y 316.453,Z 567.675,A -85,B 0,C 180,E1 -16953.943,E2 -16953.943} C_VEL
LIN {X 0,Y 315.448,Z 564.271,A -85,B 0,C 180,E1 -16954.658,E2 -16954.658} C_VEL
LIN {X 0,Y 313.081,Z 558.454,A -85,B 0,C 180,E1 -16956.312,E2 -16956.312} C_VEL
LIN {X 0,Y 311.408,Z 554.326,A -85,B 0,C 180,E1 -16957.824,E2 -16957.824} C_VEL
LIN {X 0,Y 311.171,Z 551.052,A -85,B 0,C 180,E1 -16959.833,E2 -16959.833} C_VEL
LIN {X 0,Y 311.007,Z 548.88,A -85,B 0,C 180,E1 -16961.779,E2 -16961.779} C_VEL
LIN {X 0,Y 311.156,Z 547.065,A -85,B 0,C 180,E1 -16964.442,E2 -16964.442} C_VEL
LIN {X 0,Y 311.51,Z 546.695,A -85,B 0,C 180,E1 -16966.216,E2 -16966.216} C_VEL
LIN {X 0,Y 312.208,Z 546.991,A -85,B 0,C 180,E1 -16967.975,E2 -16967.975} C_VEL
LIN {X 0,Y 313.191,Z 547.938,A -85,B 0,C 180,E1 -16969.726,E2 -16969.726} C_VEL
LIN {X 0,Y 314.543,Z 549.508,A -85,B 0,C 180,E1 -16971.446,E2 -16971.446} C_VEL
LIN {X 0,Y 316.152,Z 551.969,A -85,B 0,C 180,E1 -16973.156,E2 -16973.156} C_VEL
LIN {X 0,Y 316.539,Z 552.713,A -85,B 0,C 180,E1 -16973.564,E2 -16973.564} C_VEL
LIN {X 0,Y 316.831,Z 555.378,A -85,B 0,C 180,E1 -16974.367,E2 -16974.367} C_VEL
LIN {X 0,Y 317.193,Z 558.371,A -85,B 0,C 180,E1 -16975.1,E2 -16975.1} C_VEL
LIN {X 0,Y 318.412,Z 562.75,A -85,B 0,C 180,E1 -16975.969,E2 -16975.969} C_VEL
LIN {X 0,Y 318.17,Z 571.252,A -85,B 0,C 180,E1 -16976.666,E2 -16976.666} C_VEL
LIN {X 0,Y 306.427,Z 662.588,A -85,B 0,C 180,E1 -16980.69,E2 -16980.69} C_VEL
LIN {X 0,Y 304.262,Z 681.494,A -85,B 0,C 180,E1 -16981.614,E2 -16981.614} C_VEL
LIN {X 0,Y 302.081,Z 695.151,A -85,B 0,C 180,E1 -16982.552,E2 -16982.552} C_VEL
LIN {X 0,Y 299.757,Z 708.033,A -85,B 0,C 180,E1 -16983.734,E2 -16983.734} C_VEL
LIN {X 0,Y 297.181,Z 720.412,A -85,B 0,C 180,E1 -16985.18,E2 -16985.18} C_VEL
LIN {X 0,Y 294.204,Z 732.667,A -85,B 0,C 180,E1 -16986.973,E2 -16986.973} C_VEL
LIN {X 0,Y 291.608,Z 742.677,A -85,B 0,C 180,E1 -16988.807,E2 -16988.807} C_VEL
LIN {X 0,Y 288.832,Z 752.986,A -85,B 0,C 180,E1 -16991.192,E2 -16991.192} C_VEL
LIN {X 0,Y 286.95,Z 760.061,A -85,B 0,C 180,E1 -16993.275,E2 -16993.275} C_VEL
LIN {X 0,Y 285.147,Z 766.7,A -85,B 0,C 180,E1 -16995.731,E2 -16995.731} C_VEL
LIN {X 0,Y 284.03,Z 771.117,A -85,B 0,C 180,E1 -16997.859,E2 -16997.859} C_VEL
LIN {X 0,Y 283.204,Z 774.479,A -85,B 0,C 180,E1 -16999.996,E2 -16999.996} C_VEL
LIN {X 0,Y 282.836,Z 776.187,A -85,B 0,C 180,E1 -17001.426,E2 -17001.426} C_VEL
LIN {X 0,Y 282.571,Z 777.422,A -85,B 0,C 180,E1 -17002.856,E2 -17002.856} C_VEL
LIN {X 0,Y 282.4,Z 778.341,A -85,B 0,C 180,E1 -17004.543,E2 -17004.543} C_VEL
LIN {X 0,Y 282.398,Z 778.603,A -85,B 0,C 180,E1 -17007.147,E2 -17007.147} C_VEL
LIN {X 0,Y 282.39,Z 777.81,A -85,B 0,C 180,E1 -17009.287,E2 -17009.287} C_VEL
LIN {X 0,Y 282.352,Z 779.09,A -85,B 0,C 180,E1 -17011.426,E2 -17011.426} C_VEL
LIN {X 0,Y 282.381,Z 779.447,A -85,B 0,C 180,E1 -17012.853,E2 -17012.853} C_VEL
LIN {X 0,Y 282.384,Z 779.05,A -85,B 0,C 180,E1 -17015.714,E2 -17015.714} C_VEL
LIN {X 0,Y 282.77,Z 777.216,A -85,B 0,C 180,E1 -17018.576,E2 -17018.576} C_VEL
LIN {X 0,Y 283.612,Z 773.941,A -85,B 0,C 180,E1 -17021.434,E2 -17021.434} C_VEL
LIN {X 0,Y 284.617,Z 770.494,A -85,B 0,C 180,E1 -17023.567,E2 -17023.567} C_VEL
LIN {X 0,Y 285.996,Z 766.165,A -85,B 0,C 180,E1 -17025.683,E2 -17025.683} C_VEL
LIN {X 0,Y 288.038,Z 759.855,A -85,B 0,C 180,E1 -17028.125,E2 -17028.125} C_VEL
LIN {X 0,Y 290.541,Z 752.07,A -85,B 0,C 180,E1 -17030.533,E2 -17030.533} C_VEL
LIN {X 0,Y 293.697,Z 742.547,A -85,B 0,C 180,E1 -17032.883,E2 -17032.883} C_VEL
LIN {X 0,Y 296.849,Z 732.708,A -85,B 0,C 180,E1 -17034.85,E2 -17034.85} C_VEL
LIN {X 0,Y 300.17,Z 721.899,A -85,B 0,C 180,E1 -17036.599,E2 -17036.599} C_VEL
LIN {X 0,Y 303.712,Z 709.309,A -85,B 0,C 180,E1 -17038.243,E2 -17038.243} C_VEL
LIN {X 0,Y 307.068,Z 695.752,A -85,B 0,C 180,E1 -17039.666,E2 -17039.666} C_VEL
LIN {X 0,Y 310.095,Z 682.105,A -85,B 0,C 180,E1 -17040.755,E2 -17040.755} C_VEL
LIN {X 0,Y 312.833,Z 667.056,A -85,B 0,C 180,E1 -17041.678,E2 -17041.678} C_VEL
LIN {X 0,Y 315.111,Z 650.219,A -85,B 0,C 180,E1 -17042.41,E2 -17042.41} C_VEL
LIN {X 0,Y 321.396,Z 600.882,A -85,B 0,C 180,E1 -17044.317,E2 -17044.317} C_VEL
LIN {X 0,Y 325.06,Z 573.967,A -85,B 0,C 180,E1 -17045.386,E2 -17045.386} C_VEL
LIN {X 0,Y 322.053,Z 567.151,A -85,B 0,C 180,E1 -17047.065,E2 -17047.065} C_VEL
LIN {X 0,Y 319.628,Z 562.757,A -85,B 0,C 180,E1 -17048.564,E2 -17048.564} C_VEL
LIN {X 0,Y 317.166,Z 558.597,A -85,B 0,C 180,E1 -17050.473,E2 -17050.473} C_VEL
LIN {X 0,Y 314.562,Z 554.72,A -85,B 0,C 180,E1 -17053.444,E2 -17053.444} C_VEL
LIN {X 0,Y 313.846,Z 553.975,A -85,B 0,C 180,E1 -17054.91,E2 -17054.91} C_VEL
LIN {X 0,Y 313.473,Z 553.972,A -85,B 0,C 180,E1 -17057.242,E2 -17057.242} C_VEL
LIN {X 0,Y 314.097,Z 555.18,A -85,B 0,C 180,E1 -17059.543,E2 -17059.543} C_VEL
LIN {X 0,Y 314.769,Z 556.851,A -85,B 0,C 180,E1 -17060.85,E2 -17060.85} C_VEL
LIN {X 0,Y 317.286,Z 561.847,A -85,B 0,C 180,E1 -17063.673,E2 -17063.673} C_VEL
LIN {X 0,Y 319.618,Z 567.252,A -85,B 0,C 180,E1 -17065.549,E2 -17065.549} C_VEL
LIN {X 0,Y 321.639,Z 572.482,A -85,B 0,C 180,E1 -17066.957,E2 -17066.957} C_VEL
LIN {X 0,Y 322.018,Z 574.356,A -85,B 0,C 180,E1 -17067.273,E2 -17067.273} C_VEL
LIN {X 0,Y 322.582,Z 583.819,A -85,B 0,C 180,E1 -17068.373,E2 -17068.373} C_VEL
LIN {X 0,Y 322.742,Z 589.431,A -85,B 0,C 180,E1 -17068.927,E2 -17068.927} C_VEL
LIN {X 0,Y 312.565,Z 660.396,A -85,B 0,C 180,E1 -17072.006,E2 -17072.006} C_VEL
LIN {X 0,Y 310.055,Z 674.233,A -85,B 0,C 180,E1 -17072.86,E2 -17072.86} C_VEL
LIN {X 0,Y 306.669,Z 690,A -85,B 0,C 180,E1 -17074.187,E2 -17074.187} C_VEL
LIN {X 0,Y 303.612,Z 702.45,A -85,B 0,C 180,E1 -17075.558,E2 -17075.558} C_VEL
LIN {X 0,Y 300.407,Z 713.833,A -85,B 0,C 180,E1 -17077.111,E2 -17077.111} C_VEL
LIN {X 0,Y 297.255,Z 724.227,A -85,B 0,C 180,E1 -17078.866,E2 -17078.866} C_VEL
LIN {X 0,Y 294.13,Z 733.579,A -85,B 0,C 180,E1 -17080.819,E2 -17080.819} C_VEL
LIN {X 0,Y 291.515,Z 741.284,A -85,B 0,C 180,E1 -17082.823,E2 -17082.823} C_VEL
LIN {X 0,Y 288.967,Z 748.458,A -85,B 0,C 180,E1 -17085.204,E2 -17085.204} C_VEL
LIN {X 0,Y 286.982,Z 753.357,A -85,B 0,C 180,E1 -17087.267,E2 -17087.267} C_VEL
LIN {X 0,Y 285.61,Z 757.165,A -85,B 0,C 180,E1 -17089.365,E2 -17089.365} C_VEL
LIN {X 0,Y 284.423,Z 759.969,A -85,B 0,C 180,E1 -17091.474,E2 -17091.474} C_VEL
LIN {X 0,Y 283.266,Z 762.189,A -85,B 0,C 180,E1 -17094.304,E2 -17094.304} C_VEL
LIN {X 0,Y 282.948,Z 762.692,A -85,B 0,C 180,E1 -17095.727,E2 -17095.727} C_VEL
LIN {X 0,Y 282.686,Z 762.773,A -85,B 0,C 180,E1 -17097.15,E2 -17097.15} C_VEL
LIN {X 0,Y 282.487,Z 762.403,A -85,B 0,C 180,E1 -17098.574,E2 -17098.574} C_VEL
LIN {X 0,Y 282.388,Z 761.621,A -85,B 0,C 180,E1 -17100,E2 -17100} C_VEL
LIN {X 0,Y 282.375,Z 760.427,A -85,B 0,C 180,E1 -17101.426,E2 -17101.426} C_VEL
LIN {X 0,Y 282.383,Z 757.768,A -85,B 0,C 180,E1 -17103.567,E2 -17103.567} C_VEL
LIN {X 0,Y 282.489,Z 754.046,A -85,B 0,C 180,E1 -17105.711,E2 -17105.711} C_VEL
LIN {X 0,Y 282.742,Z 749.162,A -85,B 0,C 180,E1 -17107.858,E2 -17107.858} C_VEL
LIN {X 0,Y 283.127,Z 742.984,A -85,B 0,C 180,E1 -17110.006,E2 -17110.006} C_VEL
LIN {X 0,Y 283.743,Z 735.288,A -85,B 0,C 180,E1 -17112.154,E2 -17112.154} C_VEL
LIN {X 0,Y 284.491,Z 727.517,A -85,B 0,C 180,E1 -17113.937,E2 -17113.937} C_VEL
LIN {X 0,Y 285.17,Z 718.116,A -85,B 0,C 180,E1 -17115.729,E2 -17115.729} C_VEL
LIN {X 0,Y 286.419,Z 706.783,A -85,B 0,C 180,E1 -17117.493,E2 -17117.493} C_VEL
LIN {X 0,Y 287.595,Z 693.996,A -85,B 0,C 180,E1 -17119.077,E2 -17119.077} C_VEL
LIN {X 0,Y 288.612,Z 681.58,A -85,B 0,C 180,E1 -17120.304,E2 -17120.304} C_VEL
LIN {X 0,Y 289.536,Z 667.662,A -85,B 0,C 180,E1 -17121.352,E2 -17121.352} C_VEL
LIN {X 0,Y 290.351,Z 653.377,A -85,B 0,C 180,E1 -17122.129,E2 -17122.129} C_VEL
LIN {X 0,Y 293.795,Z 577.4,A -85,B 0,C 180,E1 -17124.984,E2 -17124.984} C_VEL
LIN {X 0,Y 289.889,Z 543.856,A -85,B 0,C 180,E1 -17126.529,E2 -17126.529} C_VEL
LIN {X 0,Y 289.497,Z 538.587,A -85,B 0,C 180,E1 -17126.806,E2 -17126.806} C_VEL
LIN {X 0,Y 290.652,Z 530.301,A -85,B 0,C 180,E1 -17128.921,E2 -17128.921} C_VEL
LIN {X 0,Y 289.846,Z 525.395,A -85,B 0,C 180,E1 -17130.283,E2 -17130.283} C_VEL
LIN {X 0,Y 286.911,Z 511.543,A -85,B 0,C 180,E1 -17134.291,E2 -17134.291} C_VEL
LIN {X 0,Y 284.365,Z 500.186,A -85,B 0,C 180,E1 -17137.808,E2 -17137.808} C_VEL
LIN {X 0,Y 284.284,Z 500.196,A -85,B 0,C 180,E1 -17142.127,E2 -17142.127} C_VEL
LIN {X 0,Y 284.257,Z 500.2,A -85,B 0,C 180,E1 -17146.189,E2 -17146.189} C_VEL
LIN {X 0,Y 284.308,Z 500.194,A -85,B 0,C 180,E1 -17150.024,E2 -17150.024} C_VEL
LIN {X 0,Y 284.334,Z 500.193,A -85,B 0,C 180,E1 -17153.614,E2 -17153.614} C_VEL
LIN {X 0,Y 284.31,Z 500.194,A -85,B 0,C 180,E1 -17157.189,E2 -17157.189} C_VEL
LIN {X 0,Y 284.36,Z 500.186,A -85,B 0,C 180,E1 -17160.376,E2 -17160.376} C_VEL
LIN {X 0,Y 284.379,Z 500.187,A -85,B 0,C 180,E1 -17163.587,E2 -17163.587} C_VEL
LIN {X 0,Y 284.368,Z 500.185,A -85,B 0,C 180,E1 -17166.707,E2 -17166.707} C_VEL
LIN {X 0,Y 284.406,Z 500.183,A -85,B 0,C 180,E1 -17171.262,E2 -17171.262} C_VEL
LIN {X 0,Y 284.493,Z 500.169,A -85,B 0,C 180,E1 -17174.459,E2 -17174.459} C_VEL
LIN {X 0,Y 284.49,Z 500.17,A -85,B 0,C 180,E1 -17178.601,E2 -17178.601} C_VEL
LIN {X 0,Y 284.661,Z 500.152,A -85,B 0,C 180,E1 -17181.481,E2 -17181.481} C_VEL
LIN {X 0,Y 284.604,Z 500.156,A -85,B 0,C 180,E1 -17184.331,E2 -17184.331} C_VEL
LIN {X 0,Y 284.86,Z 500.123,A -85,B 0,C 180,E1 -17188.586,E2 -17188.586} C_VEL
LIN {X 0,Y 284.858,Z 500.128,A -85,B 0,C 180,E1 -17191.414,E2 -17191.414} C_VEL
LIN {X 0,Y 284.699,Z 500.146,A -85,B 0,C 180,E1 -17197.09,E2 -17197.09} C_VEL
LIN {X 0,Y 284.568,Z 500.161,A -85,B 0,C 180,E1 -17199.955,E2 -17199.955} C_VEL
LIN {X 0,Y 284.483,Z 500.171,A -85,B 0,C 180,E1 -17204.303,E2 -17204.303} C_VEL
LIN {X 0,Y 284.427,Z 500.18,A -85,B 0,C 180,E1 -17207.248,E2 -17207.248} C_VEL
LIN {X 0,Y 284.38,Z 500.184,A -85,B 0,C 180,E1 -17210.242,E2 -17210.242} C_VEL
LIN {X 0,Y 284.37,Z 500.185,A -85,B 0,C 180,E1 -17213.875,E2 -17213.875} C_VEL
LIN {X 0,Y 284.395,Z 500.184,A -85,B 0,C 180,E1 -17217.173,E2 -17217.173} C_VEL
LIN {X 0,Y 284.294,Z 500.199,A -85,B 0,C 180,E1 -17221.275,E2 -17221.275} C_VEL
LIN {X 0,Y 284.363,Z 500.19,A -85,B 0,C 180,E1 -17225.354,E2 -17225.354} C_VEL
LIN {X 0,Y 284.324,Z 500.191,A -85,B 0,C 180,E1 -17228.167,E2 -17228.167} C_VEL
LIN {X 0,Y 284.27,Z 500.196,A -85,B 0,C 180,E1 -17232.125,E2 -17232.125} C_VEL
LIN {X 0,Y 284.269,Z 500.197,A -85,B 0,C 180,E1 -17236.192,E2 -17236.192} C_VEL
LIN {X 0,Y 284.307,Z 500.194,A -85,B 0,C 180,E1 -17240.024,E2 -17240.024} C_VEL
LIN {X 0,Y 284.334,Z 500.193,A -85,B 0,C 180,E1 -17243.614,E2 -17243.614} C_VEL
LIN {X 0,Y 284.335,Z 500.257,A -85,B 0,C 180,E1 -17245.047,E2 -17245.047} C_VEL
LIN {X 0,Y 288.297,Z 517.377,A -85,B 0,C 180,E1 -17248.946,E2 -17248.946} C_VEL
LIN {X 0,Y 290.752,Z 528.865,A -85,B 0,C 180,E1 -17251.485,E2 -17251.485} C_VEL
LIN {X 0,Y 290.468,Z 534.525,A -85,B 0,C 180,E1 -17252.631,E2 -17252.631} C_VEL
LIN {X 0,Y 289.143,Z 549.654,A -85,B 0,C 180,E1 -17255.647,E2 -17255.647} C_VEL
LIN {X 0,Y 291.363,Z 571.862,A -85,B 0,C 180,E1 -17256.611,E2 -17256.611} C_VEL
LIN {X 0,Y 292.282,Z 579.937,A -85,B 0,C 180,E1 -17256.958,E2 -17256.958} C_VEL
LIN {X 0,Y 289.889,Z 644.079,A -85,B 0,C 180,E1 -17259.275,E2 -17259.275} C_VEL
LIN {X 0,Y 288.999,Z 649.846,A -85,B 0,C 180,E1 -17259.459,E2 -17259.459} C_VEL
LIN {X 0,Y 285.636,Z 659.102,A -85,B 0,C 180,E1 -17259.73,E2 -17259.73} C_VEL
LIN {X 0,Y 282.381,Z 668.267,A -85,B 0,C 180,E1 -17260.124,E2 -17260.124} C_VEL
LIN {X 0,Y 281.534,Z 673.885,A -85,B 0,C 180,E1 -17260.461,E2 -17260.461} C_VEL
LIN {X 0,Y 280.605,Z 687.904,A -85,B 0,C 180,E1 -17261.567,E2 -17261.567} C_VEL
LIN {X 0,Y 279.627,Z 700.668,A -85,B 0,C 180,E1 -17262.897,E2 -17262.897} C_VEL
LIN {X 0,Y 278.702,Z 712.458,A -85,B 0,C 180,E1 -17264.459,E2 -17264.459} C_VEL
LIN {X 0,Y 277.826,Z 722.444,A -85,B 0,C 180,E1 -17266.095,E2 -17266.095} C_VEL
LIN {X 0,Y 276.968,Z 731.58,A -85,B 0,C 180,E1 -17267.916,E2 -17267.916} C_VEL
LIN {X 0,Y 276.243,Z 740.559,A -85,B 0,C 180,E1 -17270.112,E2 -17270.112} C_VEL
LIN {X 0,Y 275.749,Z 747.715,A -85,B 0,C 180,E1 -17272.31,E2 -17272.31} C_VEL
LIN {X 0,Y 275.485,Z 752.784,A -85,B 0,C 180,E1 -17274.238,E2 -17274.238} C_VEL
LIN {X 0,Y 275.389,Z 757.164,A -85,B 0,C 180,E1 -17276.342,E2 -17276.342} C_VEL
LIN {X 0,Y 275.275,Z 760.601,A -85,B 0,C 180,E1 -17278.537,E2 -17278.537} C_VEL
LIN {X 0,Y 275.276,Z 762.323,A -85,B 0,C 180,E1 -17280,E2 -17280} C_VEL
LIN {X 0,Y 275.322,Z 763.564,A -85,B 0,C 180,E1 -17281.463,E2 -17281.463} C_VEL
LIN {X 0,Y 275.433,Z 764.366,A -85,B 0,C 180,E1 -17282.925,E2 -17282.925} C_VEL
LIN {X 0,Y 275.628,Z 764.757,A -85,B 0,C 180,E1 -17284.387,E2 -17284.387} C_VEL
LIN {X 0,Y 275.977,Z 764.711,A -85,B 0,C 180,E1 -17285.847,E2 -17285.847} C_VEL
LIN {X 0,Y 276.542,Z 764.048,A -85,B 0,C 180,E1 -17287.63,E2 -17287.63} C_VEL
LIN {X 0,Y 277.49,Z 762.013,A -85,B 0,C 180,E1 -17290.212,E2 -17290.212} C_VEL
LIN {X 0,Y 278.791,Z 759.182,A -85,B 0,C 180,E1 -17292.373,E2 -17292.373} C_VEL
LIN {X 0,Y 280.298,Z 755.363,A -85,B 0,C 180,E1 -17294.521,E2 -17294.521} C_VEL
LIN {X 0,Y 282.34,Z 750.359,A -85,B 0,C 180,E1 -17296.634,E2 -17296.634} C_VEL
LIN {X 0,Y 285.177,Z 742.894,A -85,B 0,C 180,E1 -17299.059,E2 -17299.059} C_VEL
LIN {X 0,Y 288.054,Z 734.939,A -85,B 0,C 180,E1 -17301.092,E2 -17301.092} C_VEL
LIN {X 0,Y 291.232,Z 725.209,A -85,B 0,C 180,E1 -17303.05,E2 -17303.05} C_VEL
LIN {X 0,Y 294.35,Z 714.658,A -85,B 0,C 180,E1 -17304.773,E2 -17304.773} C_VEL
LIN {X 0,Y 297.137,Z 704.162,A -85,B 0,C 180,E1 -17306.138,E2 -17306.138} C_VEL
LIN {X 0,Y 299.976,Z 692.122,A -85,B 0,C 180,E1 -17307.373,E2 -17307.373} C_VEL
LIN {X 0,Y 302.792,Z 677.916,A -85,B 0,C 180,E1 -17308.507,E2 -17308.507} C_VEL
LIN {X 0,Y 305.12,Z 662.875,A -85,B 0,C 180,E1 -17309.353,E2 -17309.353} C_VEL
LIN {X 0,Y 314.482,Z 592.431,A -85,B 0,C 180,E1 -17312.34,E2 -17312.34} C_VEL
LIN {X 0,Y 313.874,Z 582.04,A -85,B 0,C 180,E1 -17313.47,E2 -17313.47} C_VEL
LIN {X 0,Y 313.056,Z 571.683,A -85,B 0,C 180,E1 -17314.814,E2 -17314.814} C_VEL
LIN {X 0,Y 310.808,Z 565.167,A -85,B 0,C 180,E1 -17316.571,E2 -17316.571} C_VEL
LIN {X 0,Y 308.697,Z 559.973,A -85,B 0,C 180,E1 -17318.548,E2 -17318.548} C_VEL
LIN {X 0,Y 307.063,Z 555.927,A -85,B 0,C 180,E1 -17320.738,E2 -17320.738} C_VEL
LIN {X 0,Y 306.802,Z 554.818,A -85,B 0,C 180,E1 -17321.63,E2 -17321.63} C_VEL
LIN {X 0,Y 306.919,Z 553.44,A -85,B 0,C 180,E1 -17323.39,E2 -17323.39} C_VEL
LIN {X 0,Y 307.264,Z 552.722,A -85,B 0,C 180,E1 -17325.158,E2 -17325.158} C_VEL
LIN {X 0,Y 307.84,Z 552.686,A -85,B 0,C 180,E1 -17326.934,E2 -17326.934} C_VEL
LIN {X 0,Y 308.695,Z 553.313,A -85,B 0,C 180,E1 -17328.704,E2 -17328.704} C_VEL
LIN {X 0,Y 310.046,Z 554.731,A -85,B 0,C 180,E1 -17330.603,E2 -17330.603} C_VEL
LIN {X 0,Y 312.022,Z 557.373,A -85,B 0,C 180,E1 -17332.706,E2 -17332.706} C_VEL
LIN {X 0,Y 313.058,Z 559.212,A -85,B 0,C 180,E1 -17333.434,E2 -17333.434} C_VEL
LIN {X 0,Y 314.884,Z 566.594,A -85,B 0,C 180,E1 -17335.06,E2 -17335.06} C_VEL
LIN {X 0,Y 314.596,Z 572.878,A -85,B 0,C 180,E1 -17335.589,E2 -17335.589} C_VEL
LIN {X 0,Y 302.28,Z 661.385,A -85,B 0,C 180,E1 -17339.568,E2 -17339.568} C_VEL
LIN {X 0,Y 299.813,Z 680.594,A -85,B 0,C 180,E1 -17340.51,E2 -17340.51} C_VEL
LIN {X 0,Y 297.259,Z 695.223,A -85,B 0,C 180,E1 -17341.528,E2 -17341.528} C_VEL
LIN {X 0,Y 294.824,Z 707.613,A -85,B 0,C 180,E1 -17342.685,E2 -17342.685} C_VEL
LIN {X 0,Y 291.983,Z 719.854,A -85,B 0,C 180,E1 -17344.134,E2 -17344.134} C_VEL
LIN {X 0,Y 289.02,Z 731.101,A -85,B 0,C 180,E1 -17345.773,E2 -17345.773} C_VEL
LIN {X 0,Y 286.145,Z 741.233,A -85,B 0,C 180,E1 -17347.623,E2 -17347.623} C_VEL
LIN {X 0,Y 283.496,Z 750.357,A -85,B 0,C 180,E1 -17349.692,E2 -17349.692} C_VEL
LIN {X 0,Y 280.874,Z 758.847,A -85,B 0,C 180,E1 -17352.108,E2 -17352.108} C_VEL
LIN {X 0,Y 279.326,Z 763.983,A -85,B 0,C 180,E1 -17353.933,E2 -17353.933} C_VEL
LIN {X 0,Y 277.895,Z 768.896,A -85,B 0,C 180,E1 -17356.098,E2 -17356.098} C_VEL
LIN {X 0,Y 276.752,Z 772.75,A -85,B 0,C 180,E1 -17358.278,E2 -17358.278} C_VEL
LIN {X 0,Y 276.185,Z 774.762,A -85,B 0,C 180,E1 -17359.739,E2 -17359.739} C_VEL
LIN {X 0,Y 275.793,Z 776.295,A -85,B 0,C 180,E1 -17361.205,E2 -17361.205} C_VEL
LIN {X 0,Y 275.505,Z 777.425,A -85,B 0,C 180,E1 -17362.672,E2 -17362.672} C_VEL
LIN {X 0,Y 275.315,Z 778.274,A -85,B 0,C 180,E1 -17364.598,E2 -17364.598} C_VEL
LIN {X 0,Y 275.323,Z 778.259,A -85,B 0,C 180,E1 -17367.074,E2 -17367.074} C_VEL
LIN {X 0,Y 275.312,Z 777.272,A -85,B 0,C 180,E1 -17369.269,E2 -17369.269} C_VEL
LIN {X 0,Y 275.277,Z 778.658,A -85,B 0,C 180,E1 -17371.463,E2 -17371.463} C_VEL
LIN {X 0,Y 275.307,Z 779.123,A -85,B 0,C 180,E1 -17372.927,E2 -17372.927} C_VEL
LIN {X 0,Y 275.297,Z 778.915,A -85,B 0,C 180,E1 -17375.861,E2 -17375.861} C_VEL
LIN {X 0,Y 275.71,Z 777.253,A -85,B 0,C 180,E1 -17378.798,E2 -17378.798} C_VEL
LIN {X 0,Y 276.633,Z 774.165,A -85,B 0,C 180,E1 -17381.727,E2 -17381.727} C_VEL
LIN {X 0,Y 277.713,Z 770.914,A -85,B 0,C 180,E1 -17383.911,E2 -17383.911} C_VEL
LIN {X 0,Y 279.697,Z 765.14,A -85,B 0,C 180,E1 -17386.796,E2 -17386.796} C_VEL
LIN {X 0,Y 282.46,Z 757.661,A -85,B 0,C 180,E1 -17389.627,E2 -17389.627} C_VEL
LIN {X 0,Y 284.881,Z 750.767,A -85,B 0,C 180,E1 -17391.719,E2 -17391.719} C_VEL
LIN {X 0,Y 287.845,Z 742.563,A -85,B 0,C 180,E1 -17393.757,E2 -17393.757} C_VEL
LIN {X 0,Y 291.233,Z 732.84,A -85,B 0,C 180,E1 -17395.746,E2 -17395.746} C_VEL
LIN {X 0,Y 294.747,Z 722.219,A -85,B 0,C 180,E1 -17397.515,E2 -17397.515} C_VEL
LIN {X 0,Y 298.375,Z 710.351,A -85,B 0,C 180,E1 -17399.108,E2 -17399.108} C_VEL
LIN {X 0,Y 302.02,Z 696.801,A -85,B 0,C 180,E1 -17400.581,E2 -17400.581} C_VEL
LIN {X 0,Y 305.032,Z 684.548,A -85,B 0,C 180,E1 -17401.612,E2 -17401.612} C_VEL
LIN {X 0,Y 307.906,Z 670.358,A -85,B 0,C 180,E1 -17402.535,E2 -17402.535} C_VEL
LIN {X 0,Y 310.531,Z 653.453,A -85,B 0,C 180,E1 -17403.336,E2 -17403.336} C_VEL
LIN {X 0,Y 319.297,Z 590.886,A -85,B 0,C 180,E1 -17405.804,E2 -17405.804} C_VEL
LIN {X 0,Y 321.23,Z 577.803,A -85,B 0,C 180,E1 -17406.336,E2 -17406.336} C_VEL
LIN {X 0,Y 318.748,Z 572.095,A -85,B 0,C 180,E1 -17407.889,E2 -17407.889} C_VEL
LIN {X 0,Y 317.159,Z 568.966,A -85,B 0,C 180,E1 -17409.001,E2 -17409.001} C_VEL
LIN {X 0,Y 314.979,Z 565.086,A -85,B 0,C 180,E1 -17410.826,E2 -17410.826} C_VEL
LIN {X 0,Y 312.694,Z 561.462,A -85,B 0,C 180,E1 -17413.649,E2 -17413.649} C_VEL
LIN {X 0,Y 311.855,Z 560.753,A -85,B 0,C 180,E1 -17415.683,E2 -17415.683} C_VEL
LIN {X 0,Y 311.858,Z 561.236,A -85,B 0,C 180,E1 -17418.318,E2 -17418.318} C_VEL
LIN {X 0,Y 312.523,Z 562.784,A -85,B 0,C 180,E1 -17420.126,E2 -17420.126} C_VEL
LIN {X 0,Y 314.863,Z 567.93,A -85,B 0,C 180,E1 -17423.175,E2 -17423.175} C_VEL
LIN {X 0,Y 316.911,Z 573.31,A -85,B 0,C 180,E1 -17425.077,E2 -17425.077} C_VEL
LIN {X 0,Y 318.578,Z 577.87,A -85,B 0,C 180,E1 -17426.339,E2 -17426.339} C_VEL
LIN {X 0,Y 318.904,Z 586.185,A -85,B 0,C 180,E1 -17427.362,E2 -17427.362} C_VEL
LIN {X 0,Y 318.922,Z 591.546,A -85,B 0,C 180,E1 -17427.893,E2 -17427.893} C_VEL
LIN {X 0,Y 308.32,Z 660.318,A -85,B 0,C 180,E1 -17430.935,E2 -17430.935} C_VEL
LIN {X 0,Y 305.481,Z 674.957,A -85,B 0,C 180,E1 -17431.86,E2 -17431.86} C_VEL
LIN {X 0,Y 302.284,Z 688.983,A -85,B 0,C 180,E1 -17433.04,E2 -17433.04} C_VEL
LIN {X 0,Y 298.961,Z 701.484,A -85,B 0,C 180,E1 -17434.408,E2 -17434.408} C_VEL
LIN {X 0,Y 295.218,Z 714.103,A -85,B 0,C 180,E1 -17436.127,E2 -17436.127} C_VEL
LIN {X 0,Y 291.547,Z 725.188,A -85,B 0,C 180,E1 -17438.06,E2 -17438.06} C_VEL
LIN {X 0,Y 288.195,Z 734.424,A -85,B 0,C 180,E1 -17440.037,E2 -17440.037} C_VEL
LIN {X 0,Y 285.357,Z 741.959,A -85,B 0,C 180,E1 -17442.07,E2 -17442.07} C_VEL
LIN {X 0,Y 282.992,Z 748.103,A -85,B 0,C 180,E1 -17444.146,E2 -17444.146} C_VEL
LIN {X 0,Y 280.845,Z 753.137,A -85,B 0,C 180,E1 -17446.247,E2 -17446.247} C_VEL
LIN {X 0,Y 279.106,Z 757.054,A -85,B 0,C 180,E1 -17448.379,E2 -17448.379} C_VEL
LIN {X 0,Y 277.745,Z 760.135,A -85,B 0,C 180,E1 -17450.699,E2 -17450.699} C_VEL
LIN {X 0,Y 276.759,Z 761.893,A -85,B 0,C 180,E1 -17452.705,E2 -17452.705} C_VEL
LIN {X 0,Y 276.238,Z 762.688,A -85,B 0,C 180,E1 -17454.159,E2 -17454.159} C_VEL
LIN {X 0,Y 275.893,Z 763.04,A -85,B 0,C 180,E1 -17455.617,E2 -17455.617} C_VEL
LIN {X 0,Y 275.617,Z 762.978,A -85,B 0,C 180,E1 -17457.077,E2 -17457.077} C_VEL
LIN {X 0,Y 275.41,Z 762.508,A -85,B 0,C 180,E1 -17458.538,E2 -17458.538} C_VEL
LIN {X 0,Y 275.308,Z 761.626,A -85,B 0,C 180,E1 -17460,E2 -17460} C_VEL
LIN {X 0,Y 275.298,Z 760.308,A -85,B 0,C 180,E1 -17461.463,E2 -17461.463} C_VEL
LIN {X 0,Y 275.283,Z 757.489,A -85,B 0,C 180,E1 -17463.659,E2 -17463.659} C_VEL
LIN {X 0,Y 275.419,Z 753.595,A -85,B 0,C 180,E1 -17465.858,E2 -17465.858} C_VEL
LIN {X 0,Y 275.744,Z 747.487,A -85,B 0,C 180,E1 -17468.427,E2 -17468.427} C_VEL
LIN {X 0,Y 276.235,Z 740.814,A -85,B 0,C 180,E1 -17470.629,E2 -17470.629} C_VEL
LIN {X 0,Y 276.908,Z 732.567,A -85,B 0,C 180,E1 -17472.831,E2 -17472.831} C_VEL
LIN {X 0,Y 277.667,Z 724.186,A -85,B 0,C 180,E1 -17474.662,E2 -17474.662} C_VEL
LIN {X 0,Y 278.657,Z 713.49,A -85,B 0,C 180,E1 -17476.584,E2 -17476.584} C_VEL
LIN {X 0,Y 279.825,Z 701.76,A -85,B 0,C 180,E1 -17478.297,E2 -17478.297} C_VEL
LIN {X 0,Y 280.996,Z 689.441,A -85,B 0,C 180,E1 -17479.734,E2 -17479.734} C_VEL
LIN {X 0,Y 282.007,Z 675.763,A -85,B 0,C 180,E1 -17480.992,E2 -17480.992} C_VEL
LIN {X 0,Y 282.949,Z 661.305,A -85,B 0,C 180,E1 -17481.97,E2 -17481.97} C_VEL
LIN {X 0,Y 283.742,Z 647.286,A -85,B 0,C 180,E1 -17482.625,E2 -17482.625} C_VEL
LIN {X 0,Y 286.849,Z 577.679,A -85,B 0,C 180,E1 -17485.31,E2 -17485.31} C_VEL
LIN {X 0,Y 283.082,Z 544.855,A -85,B 0,C 180,E1 -17486.872,E2 -17486.872} C_VEL
LIN {X 0,Y 282.598,Z 538.622,A -85,B 0,C 180,E1 -17487.177,E2 -17487.177} C_VEL
LIN {X 0,Y 283.598,Z 530.524,A -85,B 0,C 180,E1 -17489.304,E2 -17489.304} C_VEL
LIN {X 0,Y 281.257,Z 519.213,A -85,B 0,C 180,E1 -17492.588,E2 -17492.588} C_VEL
LIN {X 0,Y 278.707,Z 507.279,A -85,B 0,C 180,E1 -17496.203,E2 -17496.203} C_VEL
LIN {X 0,Y 277.294,Z 501.065,A -85,B 0,C 180,E1 -17498.215,E2 -17498.215} C_VEL
LIN {X 0,Y 277.224,Z 501.075,A -85,B 0,C 180,E1 -17502.676,E2 -17502.676} C_VEL
LIN {X 0,Y 277.211,Z 501.078,A -85,B 0,C 180,E1 -17506.802,E2 -17506.802} C_VEL
LIN {X 0,Y 277.236,Z 501.074,A -85,B 0,C 180,E1 -17510.672,E2 -17510.672} C_VEL
LIN {X 0,Y 277.286,Z 501.067,A -85,B 0,C 180,E1 -17514.341,E2 -17514.341} C_VEL
LIN {X 0,Y 277.246,Z 501.075,A -85,B 0,C 180,E1 -17517.836,E2 -17517.836} C_VEL
LIN {X 0,Y 277.291,Z 501.069,A -85,B 0,C 180,E1 -17521.212,E2 -17521.212} C_VEL
LIN {X 0,Y 277.315,Z 501.062,A -85,B 0,C 180,E1 -17524.479,E2 -17524.479} C_VEL
LIN {X 0,Y 277.287,Z 501.071,A -85,B 0,C 180,E1 -17527.655,E2 -17527.655} C_VEL
LIN {X 0,Y 277.347,Z 501.06,A -85,B 0,C 180,E1 -17530.766,E2 -17530.766} C_VEL
LIN {X 0,Y 277.436,Z 501.052,A -85,B 0,C 180,E1 -17535.326,E2 -17535.326} C_VEL
LIN {X 0,Y 277.508,Z 501.041,A -85,B 0,C 180,E1 -17539.789,E2 -17539.789} C_VEL
LIN {X 0,Y 277.655,Z 501.021,A -85,B 0,C 180,E1 -17542.729,E2 -17542.729} C_VEL
LIN {X 0,Y 277.826,Z 500.999,A -85,B 0,C 180,E1 -17548.55,E2 -17548.55} C_VEL
LIN {X 0,Y 277.823,Z 501.005,A -85,B 0,C 180,E1 -17551.449,E2 -17551.449} C_VEL
LIN {X 0,Y 277.654,Z 501.025,A -85,B 0,C 180,E1 -17557.271,E2 -17557.271} C_VEL
LIN {X 0,Y 277.508,Z 501.04,A -85,B 0,C 180,E1 -17560.211,E2 -17560.211} C_VEL
LIN {X 0,Y 277.436,Z 501.049,A -85,B 0,C 180,E1 -17564.674,E2 -17564.674} C_VEL
LIN {X 0,Y 277.346,Z 501.063,A -85,B 0,C 180,E1 -17569.234,E2 -17569.234} C_VEL
LIN {X 0,Y 277.32,Z 501.062,A -85,B 0,C 180,E1 -17574.17,E2 -17574.17} C_VEL
LIN {X 0,Y 277.324,Z 501.066,A -85,B 0,C 180,E1 -17577.504,E2 -17577.504} C_VEL
LIN {X 0,Y 277.273,Z 501.069,A -85,B 0,C 180,E1 -17580.481,E2 -17580.481} C_VEL
LIN {X 0,Y 277.255,Z 501.071,A -85,B 0,C 180,E1 -17583.895,E2 -17583.895} C_VEL
LIN {X 0,Y 277.283,Z 501.072,A -85,B 0,C 180,E1 -17587.467,E2 -17587.467} C_VEL
LIN {X 0,Y 277.211,Z 501.081,A -85,B 0,C 180,E1 -17591.236,E2 -17591.236} C_VEL
LIN {X 0,Y 277.218,Z 501.08,A -85,B 0,C 180,E1 -17595.223,E2 -17595.223} C_VEL
LIN {X 0,Y 277.224,Z 501.079,A -85,B 0,C 180,E1 -17599.512,E2 -17599.512} C_VEL
LIN {X 0,Y 277.269,Z 501.07,A -85,B 0,C 180,E1 -17602.531,E2 -17602.531} C_VEL
LIN {X 0,Y 277.303,Z 501.074,A -85,B 0,C 180,E1 -17604.679,E2 -17604.679} C_VEL
LIN {X 0,Y 281.508,Z 519.399,A -85,B 0,C 180,E1 -17608.917,E2 -17608.917} C_VEL
LIN {X 0,Y 283.603,Z 529.165,A -85,B 0,C 180,E1 -17611.103,E2 -17611.103} C_VEL
LIN {X 0,Y 283.746,Z 533.062,A -85,B 0,C 180,E1 -17611.927,E2 -17611.927} C_VEL
LIN {X 0,Y 282.211,Z 549.847,A -85,B 0,C 180,E1 -17615.332,E2 -17615.332} C_VEL
LIN {X 0,Y 284.483,Z 572.897,A -85,B 0,C 180,E1 -17616.348,E2 -17616.348} C_VEL
LIN {X 0,Y 285.298,Z 580.93,A -85,B 0,C 180,E1 -17616.697,E2 -17616.697} C_VEL
LIN {X 0,Y 282.217,Z 660.009,A -85,B 0,C 180,E1 -17619.691,E2 -17619.691} C_VEL
LIN {X 0,Y 281.534,Z 673.885,A -85,B 0,C 180,E1 -17620.461,E2 -17620.461} C_VEL
LIN {X 0,Y 280.622,Z 679.424,A -85,B 0,C 180,E1 -17620.833,E2 -17620.833} C_VEL
LIN {X 0,Y 277.217,Z 688.137,A -85,B 0,C 180,E1 -17621.509,E2 -17621.509} C_VEL
LIN {X 0,Y 273.63,Z 696.56,A -85,B 0,C 180,E1 -17622.329,E2 -17622.329} C_VEL
LIN {X 0,Y 272.448,Z 701.657,A -85,B 0,C 180,E1 -17622.92,E2 -17622.92} C_VEL
LIN {X 0,Y 271.58,Z 712.673,A -85,B 0,C 180,E1 -17624.426,E2 -17624.426} C_VEL
LIN {X 0,Y 270.689,Z 722.665,A -85,B 0,C 180,E1 -17626.104,E2 -17626.104} C_VEL
LIN {X 0,Y 269.865,Z 731.808,A -85,B 0,C 180,E1 -17627.975,E2 -17627.975} C_VEL
LIN {X 0,Y 269.137,Z 740.745,A -85,B 0,C 180,E1 -17630.228,E2 -17630.228} C_VEL
LIN {X 0,Y 268.645,Z 747.875,A -85,B 0,C 180,E1 -17632.484,E2 -17632.484} C_VEL
LIN {X 0,Y 268.405,Z 752.508,A -85,B 0,C 180,E1 -17634.272,E2 -17634.272} C_VEL
LIN {X 0,Y 268.28,Z 758.017,A -85,B 0,C 180,E1 -17636.997,E2 -17636.997} C_VEL
LIN {X 0,Y 268.205,Z 760.318,A -85,B 0,C 180,E1 -17638.498,E2 -17638.498} C_VEL
LIN {X 0,Y 268.2,Z 762.135,A -85,B 0,C 180,E1 -17640,E2 -17640} C_VEL
LIN {X 0,Y 268.249,Z 763.52,A -85,B 0,C 180,E1 -17641.501,E2 -17641.501} C_VEL
LIN {X 0,Y 268.348,Z 764.443,A -85,B 0,C 180,E1 -17643.003,E2 -17643.003} C_VEL
LIN {X 0,Y 268.564,Z 764.927,A -85,B 0,C 180,E1 -17644.503,E2 -17644.503} C_VEL
LIN {X 0,Y 268.916,Z 765.006,A -85,B 0,C 180,E1 -17646.001,E2 -17646.001} C_VEL
LIN {X 0,Y 269.471,Z 764.591,A -85,B 0,C 180,E1 -17647.662,E2 -17647.662} C_VEL
LIN {X 0,Y 270.554,Z 762.683,A -85,B 0,C 180,E1 -17650.477,E2 -17650.477} C_VEL
LIN {X 0,Y 271.928,Z 760.087,A -85,B 0,C 180,E1 -17652.69,E2 -17652.69} C_VEL
LIN {X 0,Y 273.521,Z 756.476,A -85,B 0,C 180,E1 -17654.889,E2 -17654.889} C_VEL
LIN {X 0,Y 275.689,Z 751.752,A -85,B 0,C 180,E1 -17657.048,E2 -17657.048} C_VEL
LIN {X 0,Y 278.266,Z 745.815,A -85,B 0,C 180,E1 -17659.168,E2 -17659.168} C_VEL
LIN {X 0,Y 281.156,Z 738.449,A -85,B 0,C 180,E1 -17661.251,E2 -17661.251} C_VEL
LIN {X 0,Y 284.521,Z 729.459,A -85,B 0,C 180,E1 -17663.28,E2 -17663.28} C_VEL
LIN {X 0,Y 287.515,Z 720.684,A -85,B 0,C 180,E1 -17664.872,E2 -17664.872} C_VEL
LIN {X 0,Y 290.583,Z 710.224,A -85,B 0,C 180,E1 -17666.444,E2 -17666.444} C_VEL
LIN {X 0,Y 293.782,Z 698.691,A -85,B 0,C 180,E1 -17667.807,E2 -17667.807} C_VEL
LIN {X 0,Y 296.484,Z 687.175,A -85,B 0,C 180,E1 -17668.88,E2 -17668.88} C_VEL
LIN {X 0,Y 299.15,Z 673.624,A -85,B 0,C 180,E1 -17669.852,E2 -17669.852} C_VEL
LIN {X 0,Y 301.414,Z 658.733,A -85,B 0,C 180,E1 -17670.619,E2 -17670.619} C_VEL
LIN {X 0,Y 310.671,Z 594.65,A -85,B 0,C 180,E1 -17673.372,E2 -17673.372} C_VEL
LIN {X 0,Y 310.34,Z 584.914,A -85,B 0,C 180,E1 -17674.482,E2 -17674.482} C_VEL
LIN {X 0,Y 309.894,Z 576.45,A -85,B 0,C 180,E1 -17675.607,E2 -17675.607} C_VEL
LIN {X 0,Y 307.98,Z 570.469,A -85,B 0,C 180,E1 -17677.338,E2 -17677.338} C_VEL
LIN {X 0,Y 306.36,Z 566.104,A -85,B 0,C 180,E1 -17679.081,E2 -17679.081} C_VEL
LIN {X 0,Y 305.048,Z 562.365,A -85,B 0,C 180,E1 -17681.156,E2 -17681.156} C_VEL
LIN {X 0,Y 304.303,Z 560.024,A -85,B 0,C 180,E1 -17683.488,E2 -17683.488} C_VEL
LIN {X 0,Y 304.261,Z 559.265,A -85,B 0,C 180,E1 -17684.874,E2 -17684.874} C_VEL
LIN {X 0,Y 304.916,Z 559.164,A -85,B 0,C 180,E1 -17687.132,E2 -17687.132} C_VEL
LIN {X 0,Y 306.245,Z 560.241,A -85,B 0,C 180,E1 -17689.228,E2 -17689.228} C_VEL
LIN {X 0,Y 308.181,Z 562.114,A -85,B 0,C 180,E1 -17691.158,E2 -17691.158} C_VEL
LIN {X 0,Y 309.939,Z 564.15,A -85,B 0,C 180,E1 -17692.527,E2 -17692.527} C_VEL
LIN {X 0,Y 310.457,Z 565.488,A -85,B 0,C 180,E1 -17692.98,E2 -17692.98} C_VEL
LIN {X 0,Y 311.535,Z 570.837,A -85,B 0,C 180,E1 -17694.151,E2 -17694.151} C_VEL
LIN {X 0,Y 311.218,Z 575.232,A -85,B 0,C 180,E1 -17694.506,E2 -17694.506} C_VEL
LIN {X 0,Y 298.24,Z 661.615,A -85,B 0,C 180,E1 -17698.458,E2 -17698.458} C_VEL
LIN {X 0,Y 295.535,Z 680.418,A -85,B 0,C 180,E1 -17699.398,E2 -17699.398} C_VEL
LIN {X 0,Y 292.586,Z 695.972,A -85,B 0,C 180,E1 -17700.5,E2 -17700.5} C_VEL
LIN {X 0,Y 289.683,Z 708.942,A -85,B 0,C 180,E1 -17701.765,E2 -17701.765} C_VEL
LIN {X 0,Y 286.646,Z 720.839,A -85,B 0,C 180,E1 -17703.223,E2 -17703.223} C_VEL
LIN {X 0,Y 283.155,Z 732.702,A -85,B 0,C 180,E1 -17705.042,E2 -17705.042} C_VEL
LIN {X 0,Y 279.827,Z 743.259,A -85,B 0,C 180,E1 -17707.09,E2 -17707.09} C_VEL
LIN {X 0,Y 277.013,Z 751.884,A -85,B 0,C 180,E1 -17709.195,E2 -17709.195} C_VEL
LIN {X 0,Y 274.725,Z 758.573,A -85,B 0,C 180,E1 -17711.179,E2 -17711.179} C_VEL
LIN {X 0,Y 272.569,Z 764.855,A -85,B 0,C 180,E1 -17713.523,E2 -17713.523} C_VEL
LIN {X 0,Y 271.009,Z 769.535,A -85,B 0,C 180,E1 -17715.738,E2 -17715.738} C_VEL
LIN {X 0,Y 269.813,Z 773.143,A -85,B 0,C 180,E1 -17717.973,E2 -17717.973} C_VEL
LIN {X 0,Y 268.744,Z 776.416,A -85,B 0,C 180,E1 -17720.973,E2 -17720.973} C_VEL
LIN {X 0,Y 268.444,Z 777.442,A -85,B 0,C 180,E1 -17722.478,E2 -17722.478} C_VEL
LIN {X 0,Y 268.209,Z 778.148,A -85,B 0,C 180,E1 -17724.706,E2 -17724.706} C_VEL
LIN {X 0,Y 268.25,Z 777.903,A -85,B 0,C 180,E1 -17726.996,E2 -17726.996} C_VEL
LIN {X 0,Y 268.238,Z 776.681,A -85,B 0,C 180,E1 -17729.249,E2 -17729.249} C_VEL
LIN {X 0,Y 268.203,Z 778.184,A -85,B 0,C 180,E1 -17731.502,E2 -17731.502} C_VEL
LIN {X 0,Y 268.233,Z 778.733,A -85,B 0,C 180,E1 -17733.004,E2 -17733.004} C_VEL
LIN {X 0,Y 268.221,Z 778.721,A -85,B 0,C 180,E1 -17736.016,E2 -17736.016} C_VEL
LIN {X 0,Y 268.671,Z 777.286,A -85,B 0,C 180,E1 -17739.03,E2 -17739.03} C_VEL
LIN {X 0,Y 269.646,Z 774.419,A -85,B 0,C 180,E1 -17742.035,E2 -17742.035} C_VEL
LIN {X 0,Y 270.828,Z 771.299,A -85,B 0,C 180,E1 -17744.272,E2 -17744.272} C_VEL
LIN {X 0,Y 272.935,Z 765.834,A -85,B 0,C 180,E1 -17747.225,E2 -17747.225} C_VEL
LIN {X 0,Y 275.849,Z 758.632,A -85,B 0,C 180,E1 -17750.118,E2 -17750.118} C_VEL
LIN {X 0,Y 278.916,Z 750.805,A -85,B 0,C 180,E1 -17752.598,E2 -17752.598} C_VEL
LIN {X 0,Y 282.666,Z 741.263,A -85,B 0,C 180,E1 -17755.004,E2 -17755.004} C_VEL
LIN {X 0,Y 286.33,Z 731.402,A -85,B 0,C 180,E1 -17757.006,E2 -17757.006} C_VEL
LIN {X 0,Y 290.514,Z 719.503,A -85,B 0,C 180,E1 -17758.936,E2 -17758.936} C_VEL
LIN {X 0,Y 294.347,Z 707.671,A -85,B 0,C 180,E1 -17760.49,E2 -17760.49} C_VEL
LIN {X 0,Y 297.836,Z 695.488,A -85,B 0,C 180,E1 -17761.772,E2 -17761.772} C_VEL
LIN {X 0,Y 301.273,Z 681.997,A -85,B 0,C 180,E1 -17762.873,E2 -17762.873} C_VEL
LIN {X 0,Y 304.498,Z 666.638,A -85,B 0,C 180,E1 -17763.836,E2 -17763.836} C_VEL
LIN {X 0,Y 307.103,Z 649.652,A -85,B 0,C 180,E1 -17764.599,E2 -17764.599} C_VEL
LIN {X 0,Y 316.794,Z 586.489,A -85,B 0,C 180,E1 -17767.13,E2 -17767.13} C_VEL
LIN {X 0,Y 317.537,Z 581.577,A -85,B 0,C 180,E1 -17767.353,E2 -17767.353} C_VEL
LIN {X 0,Y 315.738,Z 577.413,A -85,B 0,C 180,E1 -17768.6,E2 -17768.6} C_VEL
LIN {X 0,Y 314.286,Z 574.474,A -85,B 0,C 180,E1 -17769.751,E2 -17769.751} C_VEL
LIN {X 0,Y 312.869,Z 571.701,A -85,B 0,C 180,E1 -17771.1,E2 -17771.1} C_VEL
LIN {X 0,Y 310.819,Z 568.148,A -85,B 0,C 180,E1 -17773.909,E2 -17773.909} C_VEL
LIN {X 0,Y 310.16,Z 567.661,A -85,B 0,C 180,E1 -17775.377,E2 -17775.377} C_VEL
LIN {X 0,Y 310.033,Z 568.011,A -85,B 0,C 180,E1 -17778.018,E2 -17778.018} C_VEL
LIN {X 0,Y 310.588,Z 569.352,A -85,B 0,C 180,E1 -17779.797,E2 -17779.797} C_VEL
LIN {X 0,Y 312.584,Z 574.441,A -85,B 0,C 180,E1 -17782.83,E2 -17782.83} C_VEL
LIN {X 0,Y 314.402,Z 579.697,A -85,B 0,C 180,E1 -17784.698,E2 -17784.698} C_VEL
LIN {X 0,Y 315.384,Z 582.838,A -85,B 0,C 180,E1 -17785.591,E2 -17785.591} C_VEL
LIN {X 0,Y 315.489,Z 592.427,A -85,B 0,C 180,E1 -17786.743,E2 -17786.743} C_VEL
LIN {X 0,Y 312.472,Z 610.836,A -85,B 0,C 180,E1 -17787.595,E2 -17787.595} C_VEL
LIN {X 0,Y 304.176,Z 661.362,A -85,B 0,C 180,E1 -17789.88,E2 -17789.88} C_VEL
LIN {X 0,Y 301.073,Z 676.195,A -85,B 0,C 180,E1 -17790.837,E2 -17790.837} C_VEL
LIN {X 0,Y 297.675,Z 689.776,A -85,B 0,C 180,E1 -17792.015,E2 -17792.015} C_VEL
LIN {X 0,Y 293.772,Z 703.343,A -85,B 0,C 180,E1 -17793.54,E2 -17793.54} C_VEL
LIN {X 0,Y 290.154,Z 714.509,A -85,B 0,C 180,E1 -17795.112,E2 -17795.112} C_VEL
LIN {X 0,Y 285.928,Z 726.341,A -85,B 0,C 180,E1 -17797.224,E2 -17797.224} C_VEL
LIN {X 0,Y 282.364,Z 735.335,A -85,B 0,C 180,E1 -17799.226,E2 -17799.226} C_VEL
LIN {X 0,Y 278.817,Z 743.798,A -85,B 0,C 180,E1 -17801.634,E2 -17801.634} C_VEL
LIN {X 0,Y 276.323,Z 749.643,A -85,B 0,C 180,E1 -17803.753,E2 -17803.753} C_VEL
LIN {X 0,Y 274.059,Z 754.357,A -85,B 0,C 180,E1 -17805.9,E2 -17805.9} C_VEL
LIN {X 0,Y 272.23,Z 758.048,A -85,B 0,C 180,E1 -17808.081,E2 -17808.081} C_VEL
LIN {X 0,Y 270.74,Z 760.965,A -85,B 0,C 180,E1 -17810.55,E2 -17810.55} C_VEL
LIN {X 0,Y 269.767,Z 762.479,A -85,B 0,C 180,E1 -17812.515,E2 -17812.515} C_VEL
LIN {X 0,Y 269.191,Z 763.116,A -85,B 0,C 180,E1 -17814.006,E2 -17814.006} C_VEL
LIN {X 0,Y 268.841,Z 763.346,A -85,B 0,C 180,E1 -17815.502,E2 -17815.502} C_VEL
LIN {X 0,Y 268.549,Z 763.177,A -85,B 0,C 180,E1 -17817,E2 -17817} C_VEL
LIN {X 0,Y 268.335,Z 762.603,A -85,B 0,C 180,E1 -17818.499,E2 -17818.499} C_VEL
LIN {X 0,Y 268.231,Z 761.579,A -85,B 0,C 180,E1 -17820,E2 -17820} C_VEL
LIN {X 0,Y 268.223,Z 760.116,A -85,B 0,C 180,E1 -17821.501,E2 -17821.501} C_VEL
LIN {X 0,Y 268.186,Z 757.095,A -85,B 0,C 180,E1 -17823.756,E2 -17823.756} C_VEL
LIN {X 0,Y 268.349,Z 752.987,A -85,B 0,C 180,E1 -17826.013,E2 -17826.013} C_VEL
LIN {X 0,Y 268.704,Z 746.682,A -85,B 0,C 180,E1 -17828.65,E2 -17828.65} C_VEL
LIN {X 0,Y 269.2,Z 739.798,A -85,B 0,C 180,E1 -17830.91,E2 -17830.91} C_VEL
LIN {X 0,Y 269.957,Z 731.188,A -85,B 0,C 180,E1 -17833.167,E2 -17833.167} C_VEL
LIN {X 0,Y 270.896,Z 720.57,A -85,B 0,C 180,E1 -17835.422,E2 -17835.422} C_VEL
LIN {X 0,Y 271.927,Z 710.109,A -85,B 0,C 180,E1 -17837.213,E2 -17837.213} C_VEL
LIN {X 0,Y 273.186,Z 697.623,A -85,B 0,C 180,E1 -17838.953,E2 -17838.953} C_VEL
LIN {X 0,Y 274.343,Z 684.137,A -85,B 0,C 180,E1 -17840.429,E2 -17840.429} C_VEL
LIN {X 0,Y 275.256,Z 671.23,A -85,B 0,C 180,E1 -17841.533,E2 -17841.533} C_VEL
LIN {X 0,Y 276.215,Z 656.73,A -85,B 0,C 180,E1 -17842.436,E2 -17842.436} C_VEL
LIN {X 0,Y 278.109,Z 617.407,A -85,B 0,C 180,E1 -17844.079,E2 -17844.079} C_VEL
LIN {X 0,Y 279.931,Z 578.075,A -85,B 0,C 180,E1 -17845.656,E2 -17845.656} C_VEL
LIN {X 0,Y 276.297,Z 546.045,A -85,B 0,C 180,E1 -17847.217,E2 -17847.217} C_VEL
LIN {X 0,Y 275.741,Z 538.417,A -85,B 0,C 180,E1 -17847.617,E2 -17847.617} C_VEL
LIN {X 0,Y 276.608,Z 532.37,A -85,B 0,C 180,E1 -17849.238,E2 -17849.238} C_VEL
LIN {X 0,Y 275.515,Z 525.973,A -85,B 0,C 180,E1 -17851.101,E2 -17851.101} C_VEL
LIN {X 0,Y 272.426,Z 511.628,A -85,B 0,C 180,E1 -17855.481,E2 -17855.481} C_VEL
LIN {X 0,Y 270.247,Z 501.942,A -85,B 0,C 180,E1 -17858.619,E2 -17858.619} C_VEL
LIN {X 0,Y 270.17,Z 501.956,A -85,B 0,C 180,E1 -17863.25,E2 -17863.25} C_VEL
LIN {X 0,Y 270.173,Z 501.958,A -85,B 0,C 180,E1 -17867.442,E2 -17867.442} C_VEL
LIN {X 0,Y 270.208,Z 501.953,A -85,B 0,C 180,E1 -17871.374,E2 -17871.374} C_VEL
LIN {X 0,Y 270.203,Z 501.95,A -85,B 0,C 180,E1 -17875.094,E2 -17875.094} C_VEL
LIN {X 0,Y 270.202,Z 501.951,A -85,B 0,C 180,E1 -17879.13,E2 -17879.13} C_VEL
LIN {X 0,Y 270.266,Z 501.942,A -85,B 0,C 180,E1 -17882.145,E2 -17882.145} C_VEL
LIN {X 0,Y 270.279,Z 501.944,A -85,B 0,C 180,E1 -17885.519,E2 -17885.519} C_VEL
LIN {X 0,Y 270.303,Z 501.937,A -85,B 0,C 180,E1 -17890.244,E2 -17890.244} C_VEL
LIN {X 0,Y 270.404,Z 501.925,A -85,B 0,C 180,E1 -17894.935,E2 -17894.935} C_VEL
LIN {X 0,Y 270.443,Z 501.923,A -85,B 0,C 180,E1 -17899.519,E2 -17899.519} C_VEL
LIN {X 0,Y 270.613,Z 501.898,A -85,B 0,C 180,E1 -17902.539,E2 -17902.539} C_VEL
LIN {X 0,Y 270.792,Z 501.875,A -85,B 0,C 180,E1 -17908.513,E2 -17908.513} C_VEL
LIN {X 0,Y 270.789,Z 501.881,A -85,B 0,C 180,E1 -17911.487,E2 -17911.487} C_VEL
LIN {X 0,Y 270.612,Z 501.902,A -85,B 0,C 180,E1 -17917.461,E2 -17917.461} C_VEL
LIN {X 0,Y 270.443,Z 501.919,A -85,B 0,C 180,E1 -17920.481,E2 -17920.481} C_VEL
LIN {X 0,Y 270.404,Z 501.926,A -85,B 0,C 180,E1 -17925.065,E2 -17925.065} C_VEL
LIN {X 0,Y 270.303,Z 501.939,A -85,B 0,C 180,E1 -17929.755,E2 -17929.755} C_VEL
LIN {X 0,Y 270.275,Z 501.94,A -85,B 0,C 180,E1 -17934.586,E2 -17934.586} C_VEL
LIN {X 0,Y 270.27,Z 501.942,A -85,B 0,C 180,E1 -17937.909,E2 -17937.909} C_VEL
LIN {X 0,Y 270.185,Z 501.956,A -85,B 0,C 180,E1 -17941.348,E2 -17941.348} C_VEL
LIN {X 0,Y 270.216,Z 501.948,A -85,B 0,C 180,E1 -17944.904,E2 -17944.904} C_VEL
LIN {X 0,Y 270.223,Z 501.948,A -85,B 0,C 180,E1 -17948.717,E2 -17948.717} C_VEL
LIN {X 0,Y 270.173,Z 501.956,A -85,B 0,C 180,E1 -17953.251,E2 -17953.251} C_VEL
LIN {X 0,Y 270.175,Z 501.957,A -85,B 0,C 180,E1 -17957.442,E2 -17957.442} C_VEL
LIN {X 0,Y 270.208,Z 501.954,A -85,B 0,C 180,E1 -17961.374,E2 -17961.374} C_VEL
LIN {X 0,Y 270.251,Z 501.982,A -85,B 0,C 180,E1 -17964.317,E2 -17964.317} C_VEL
LIN {X 0,Y 274.041,Z 518.444,A -85,B 0,C 180,E1 -17968.198,E2 -17968.198} C_VEL
LIN {X 0,Y 276.794,Z 531.391,A -85,B 0,C 180,E1 -17971.156,E2 -17971.156} C_VEL
LIN {X 0,Y 276.249,Z 539.039,A -85,B 0,C 180,E1 -17972.746,E2 -17972.746} C_VEL
LIN {X 0,Y 275.305,Z 550.222,A -85,B 0,C 180,E1 -17975.017,E2 -17975.017} C_VEL
LIN {X 0,Y 277.261,Z 571.222,A -85,B 0,C 180,E1 -17975.963,E2 -17975.963} C_VEL
LIN {X 0,Y 278.348,Z 581.232,A -85,B 0,C 180,E1 -17976.419,E2 -17976.419} C_VEL
LIN {X 0,Y 275.125,Z 661.342,A -85,B 0,C 180,E1 -17979.583,E2 -17979.583} C_VEL
LIN {X 0,Y 274.46,Z 674.671,A -85,B 0,C 180,E1 -17980.361,E2 -17980.361} C_VEL
LIN {X 0,Y 273.525,Z 688.13,A -85,B 0,C 180,E1 -17981.46,E2 -17981.46} C_VEL
LIN {X 0,Y 272.621,Z 700.065,A -85,B 0,C 180,E1 -17982.724,E2 -17982.724} C_VEL
LIN {X 0,Y 272.448,Z 701.657,A -85,B 0,C 180,E1 -17982.92,E2 -17982.92} C_VEL
LIN {X 0,Y 271.286,Z 706.67,A -85,B 0,C 180,E1 -17983.554,E2 -17983.554} C_VEL
LIN {X 0,Y 267.743,Z 714.375,A -85,B 0,C 180,E1 -17984.663,E2 -17984.663} C_VEL
LIN {X 0,Y 264.284,Z 721.623,A -85,B 0,C 180,E1 -17985.908,E2 -17985.908} C_VEL
LIN {X 0,Y 263.255,Z 725.943,A -85,B 0,C 180,E1 -17986.753,E2 -17986.753} C_VEL
LIN {X 0,Y 262.47,Z 735.058,A -85,B 0,C 180,E1 -17988.806,E2 -17988.806} C_VEL
LIN {X 0,Y 261.822,Z 743.411,A -85,B 0,C 180,E1 -17991.121,E2 -17991.121} C_VEL
LIN {X 0,Y 261.518,Z 749.079,A -85,B 0,C 180,E1 -17993.054,E2 -17993.054} C_VEL
LIN {X 0,Y 261.218,Z 754.587,A -85,B 0,C 180,E1 -17995.37,E2 -17995.37} C_VEL
LIN {X 0,Y 261.18,Z 758.817,A -85,B 0,C 180,E1 -17997.687,E2 -17997.687} C_VEL
LIN {X 0,Y 261.126,Z 761.91,A -85,B 0,C 180,E1 -18000,E2 -18000} C_VEL
LIN {X 0,Y 261.177,Z 763.387,A -85,B 0,C 180,E1 -18001.542,E2 -18001.542} C_VEL
LIN {X 0,Y 261.268,Z 764.456,A -85,B 0,C 180,E1 -18003.084,E2 -18003.084} C_VEL
LIN {X 0,Y 261.484,Z 765.097,A -85,B 0,C 180,E1 -18004.625,E2 -18004.625} C_VEL
LIN {X 0,Y 261.862,Z 765.276,A -85,B 0,C 180,E1 -18006.163,E2 -18006.163} C_VEL
LIN {X 0,Y 262.401,Z 765.051,A -85,B 0,C 180,E1 -18007.696,E2 -18007.696} C_VEL
LIN {X 0,Y 262.873,Z 764.441,A -85,B 0,C 180,E1 -18009.231,E2 -18009.231} C_VEL
LIN {X 0,Y 263.63,Z 763.38,A -85,B 0,C 180,E1 -18010.755,E2 -18010.755} C_VEL
LIN {X 0,Y 264.586,Z 761.877,A -85,B 0,C 180,E1 -18012.269,E2 -18012.269} C_VEL
LIN {X 0,Y 266.158,Z 758.861,A -85,B 0,C 180,E1 -18014.528,E2 -18014.528} C_VEL
LIN {X 0,Y 268.28,Z 754.791,A -85,B 0,C 180,E1 -18016.748,E2 -18016.748} C_VEL
LIN {X 0,Y 271.243,Z 748.573,A -85,B 0,C 180,E1 -18019.291,E2 -18019.291} C_VEL
LIN {X 0,Y 274.305,Z 741.863,A -85,B 0,C 180,E1 -18021.414,E2 -18021.414} C_VEL
LIN {X 0,Y 277.705,Z 733.595,A -85,B 0,C 180,E1 -18023.49,E2 -18023.49} C_VEL
LIN {X 0,Y 281.441,Z 723.807,A -85,B 0,C 180,E1 -18025.446,E2 -18025.446} C_VEL
LIN {X 0,Y 284.939,Z 713.253,A -85,B 0,C 180,E1 -18027.149,E2 -18027.149} C_VEL
LIN {X 0,Y 288.367,Z 701.918,A -85,B 0,C 180,E1 -18028.574,E2 -18028.574} C_VEL
LIN {X 0,Y 291.737,Z 689.173,A -85,B 0,C 180,E1 -18029.842,E2 -18029.842} C_VEL
LIN {X 0,Y 294.465,Z 676.59,A -85,B 0,C 180,E1 -18030.794,E2 -18030.794} C_VEL
LIN {X 0,Y 296.921,Z 662.555,A -85,B 0,C 180,E1 -18031.58,E2 -18031.58} C_VEL
LIN {X 0,Y 307.147,Z 596.385,A -85,B 0,C 180,E1 -18034.497,E2 -18034.497} C_VEL
LIN {X 0,Y 306.933,Z 583.141,A -85,B 0,C 180,E1 -18036.138,E2 -18036.138} C_VEL
LIN {X 0,Y 306.744,Z 580.898,A -85,B 0,C 180,E1 -18036.52,E2 -18036.52} C_VEL
LIN {X 0,Y 305.423,Z 576.38,A -85,B 0,C 180,E1 -18037.901,E2 -18037.901} C_VEL
LIN {X 0,Y 304.154,Z 572.428,A -85,B 0,C 180,E1 -18039.516,E2 -18039.516} C_VEL
LIN {X 0,Y 303.052,Z 568.718,A -85,B 0,C 180,E1 -18041.646,E2 -18041.646} C_VEL
LIN {X 0,Y 302.468,Z 566.678,A -85,B 0,C 180,E1 -18043.92,E2 -18043.92} C_VEL
LIN {X 0,Y 302.734,Z 565.989,A -85,B 0,C 180,E1 -18046.027,E2 -18046.027} C_VEL
LIN {X 0,Y 303.509,Z 566.323,A -85,B 0,C 180,E1 -18047.816,E2 -18047.816} C_VEL
LIN {X 0,Y 304.986,Z 567.608,A -85,B 0,C 180,E1 -18049.817,E2 -18049.817} C_VEL
LIN {X 0,Y 307.555,Z 570.407,A -85,B 0,C 180,E1 -18052.091,E2 -18052.091} C_VEL
LIN {X 0,Y 307.921,Z 571.927,A -85,B 0,C 180,E1 -18052.53,E2 -18052.53} C_VEL
LIN {X 0,Y 308.447,Z 574.732,A -85,B 0,C 180,E1 -18053.181,E2 -18053.181} C_VEL
LIN {X 0,Y 308.221,Z 576.857,A -85,B 0,C 180,E1 -18053.346,E2 -18053.346} C_VEL
LIN {X 0,Y 294.419,Z 662.141,A -85,B 0,C 180,E1 -18057.309,E2 -18057.309} C_VEL
LIN {X 0,Y 291.679,Z 679.493,A -85,B 0,C 180,E1 -18058.192,E2 -18058.192} C_VEL
LIN {X 0,Y 289.05,Z 692.662,A -85,B 0,C 180,E1 -18059.094,E2 -18059.094} C_VEL
LIN {X 0,Y 286.181,Z 704.667,A -85,B 0,C 180,E1 -18060.179,E2 -18060.179} C_VEL
LIN {X 0,Y 282.799,Z 717.163,A -85,B 0,C 180,E1 -18061.622,E2 -18061.622} C_VEL
LIN {X 0,Y 279.367,Z 728.496,A -85,B 0,C 180,E1 -18063.277,E2 -18063.277} C_VEL
LIN {X 0,Y 275.835,Z 738.871,A -85,B 0,C 180,E1 -18065.14,E2 -18065.14} C_VEL
LIN {X 0,Y 272.482,Z 748.173,A -85,B 0,C 180,E1 -18067.239,E2 -18067.239} C_VEL
LIN {X 0,Y 269.632,Z 755.885,A -85,B 0,C 180,E1 -18069.398,E2 -18069.398} C_VEL
LIN {X 0,Y 267.206,Z 762.18,A -85,B 0,C 180,E1 -18071.602,E2 -18071.602} C_VEL
LIN {X 0,Y 265.283,Z 767.32,A -85,B 0,C 180,E1 -18073.849,E2 -18073.849} C_VEL
LIN {X 0,Y 263.638,Z 771.366,A -85,B 0,C 180,E1 -18076.118,E2 -18076.118} C_VEL
LIN {X 0,Y 262.858,Z 773.505,A -85,B 0,C 180,E1 -18077.649,E2 -18077.649} C_VEL
LIN {X 0,Y 262.208,Z 775.232,A -85,B 0,C 180,E1 -18079.186,E2 -18079.186} C_VEL
LIN {X 0,Y 261.715,Z 776.528,A -85,B 0,C 180,E1 -18080.728,E2 -18080.728} C_VEL
LIN {X 0,Y 261.373,Z 777.385,A -85,B 0,C 180,E1 -18082.274,E2 -18082.274} C_VEL
LIN {X 0,Y 261.132,Z 777.919,A -85,B 0,C 180,E1 -18084.751,E2 -18084.751} C_VEL
LIN {X 0,Y 261.177,Z 777.513,A -85,B 0,C 180,E1 -18086.915,E2 -18086.915} C_VEL
LIN {X 0,Y 261.164,Z 776.101,A -85,B 0,C 180,E1 -18089.326,E2 -18089.326} C_VEL
LIN {X 0,Y 261.132,Z 777.699,A -85,B 0,C 180,E1 -18091.542,E2 -18091.542} C_VEL
LIN {X 0,Y 261.161,Z 778.335,A -85,B 0,C 180,E1 -18093.085,E2 -18093.085} C_VEL
LIN {X 0,Y 261.146,Z 778.506,A -85,B 0,C 180,E1 -18096.18,E2 -18096.18} C_VEL
LIN {X 0,Y 261.62,Z 777.263,A -85,B 0,C 180,E1 -18099.276,E2 -18099.276} C_VEL
LIN {X 0,Y 262.666,Z 774.629,A -85,B 0,C 180,E1 -18102.36,E2 -18102.36} C_VEL
LIN {X 0,Y 263.961,Z 771.698,A -85,B 0,C 180,E1 -18104.652,E2 -18104.652} C_VEL
LIN {X 0,Y 266.192,Z 766.487,A -85,B 0,C 180,E1 -18107.676,E2 -18107.676} C_VEL
LIN {X 0,Y 269.259,Z 759.665,A -85,B 0,C 180,E1 -18110.632,E2 -18110.632} C_VEL
LIN {X 0,Y 272.506,Z 752.173,A -85,B 0,C 180,E1 -18113.16,E2 -18113.16} C_VEL
LIN {X 0,Y 276.425,Z 743.011,A -85,B 0,C 180,E1 -18115.609,E2 -18115.609} C_VEL
LIN {X 0,Y 280.275,Z 733.617,A -85,B 0,C 180,E1 -18117.639,E2 -18117.639} C_VEL
LIN {X 0,Y 284.624,Z 722.442,A -85,B 0,C 180,E1 -18119.594,E2 -18119.594} C_VEL
LIN {X 0,Y 289.045,Z 709.8,A -85,B 0,C 180,E1 -18121.339,E2 -18121.339} C_VEL
LIN {X 0,Y 292.857,Z 697.775,A -85,B 0,C 180,E1 -18122.681,E2 -18122.681} C_VEL
LIN {X 0,Y 296.173,Z 686.083,A -85,B 0,C 180,E1 -18123.702,E2 -18123.702} C_VEL
LIN {X 0,Y 299.794,Z 670.852,A -85,B 0,C 180,E1 -18124.747,E2 -18124.747} C_VEL
LIN {X 0,Y 302.856,Z 654.367,A -85,B 0,C 180,E1 -18125.563,E2 -18125.563} C_VEL
LIN {X 0,Y 311.062,Z 603.245,A -85,B 0,C 180,E1 -18127.65,E2 -18127.65} C_VEL
LIN {X 0,Y 314.057,Z 585.662,A -85,B 0,C 180,E1 -18128.369,E2 -18128.369} C_VEL
LIN {X 0,Y 312.238,Z 581.409,A -85,B 0,C 180,E1 -18129.878,E2 -18129.878} C_VEL
LIN {X 0,Y 310.658,Z 578.164,A -85,B 0,C 180,E1 -18131.472,E2 -18131.472} C_VEL
LIN {X 0,Y 308.973,Z 575.024,A -85,B 0,C 180,E1 -18133.996,E2 -18133.996} C_VEL
LIN {X 0,Y 308.469,Z 574.598,A -85,B 0,C 180,E1 -18135.066,E2 -18135.066} C_VEL
LIN {X 0,Y 308.178,Z 574.748,A -85,B 0,C 180,E1 -18137.621,E2 -18137.621} C_VEL
LIN {X 0,Y 308.636,Z 575.977,A -85,B 0,C 180,E1 -18139.49,E2 -18139.49} C_VEL
LIN {X 0,Y 310.303,Z 580.907,A -85,B 0,C 180,E1 -18142.467,E2 -18142.467} C_VEL
LIN {X 0,Y 311.772,Z 585.685,A -85,B 0,C 180,E1 -18144.192,E2 -18144.192} C_VEL
LIN {X 0,Y 312.371,Z 588.022,A -85,B 0,C 180,E1 -18144.83,E2 -18144.83} C_VEL
LIN {X 0,Y 312.131,Z 595.471,A -85,B 0,C 180,E1 -18145.714,E2 -18145.714} C_VEL
LIN {X 0,Y 300.583,Z 661.193,A -85,B 0,C 180,E1 -18148.701,E2 -18148.701} C_VEL
LIN {X 0,Y 297.261,Z 675.873,A -85,B 0,C 180,E1 -18149.645,E2 -18149.645} C_VEL
LIN {X 0,Y 293.232,Z 690.883,A -85,B 0,C 180,E1 -18150.965,E2 -18150.965} C_VEL
LIN {X 0,Y 289.488,Z 702.956,A -85,B 0,C 180,E1 -18152.335,E2 -18152.335} C_VEL
LIN {X 0,Y 285.246,Z 715.087,A -85,B 0,C 180,E1 -18154.066,E2 -18154.066} C_VEL
LIN {X 0,Y 281.049,Z 725.983,A -85,B 0,C 180,E1 -18156.024,E2 -18156.024} C_VEL
LIN {X 0,Y 277.176,Z 735.01,A -85,B 0,C 180,E1 -18158.038,E2 -18158.038} C_VEL
LIN {X 0,Y 273.853,Z 742.478,A -85,B 0,C 180,E1 -18160.121,E2 -18160.121} C_VEL
LIN {X 0,Y 271.408,Z 747.62,A -85,B 0,C 180,E1 -18161.896,E2 -18161.896} C_VEL
LIN {X 0,Y 268.882,Z 752.783,A -85,B 0,C 180,E1 -18164.071,E2 -18164.071} C_VEL
LIN {X 0,Y 266.587,Z 756.884,A -85,B 0,C 180,E1 -18166.275,E2 -18166.275} C_VEL
LIN {X 0,Y 265.361,Z 759.052,A -85,B 0,C 180,E1 -18167.768,E2 -18167.768} C_VEL
LIN {X 0,Y 263.751,Z 761.801,A -85,B 0,C 180,E1 -18170.374,E2 -18170.374} C_VEL
LIN {X 0,Y 262.755,Z 763.016,A -85,B 0,C 180,E1 -18172.314,E2 -18172.314} C_VEL
LIN {X 0,Y 262.149,Z 763.53,A -85,B 0,C 180,E1 -18173.844,E2 -18173.844} C_VEL
LIN {X 0,Y 261.791,Z 763.648,A -85,B 0,C 180,E1 -18175.38,E2 -18175.38} C_VEL
LIN {X 0,Y 261.485,Z 763.343,A -85,B 0,C 180,E1 -18176.919,E2 -18176.919} C_VEL
LIN {X 0,Y 261.262,Z 762.603,A -85,B 0,C 180,E1 -18178.459,E2 -18178.459} C_VEL
LIN {X 0,Y 261.156,Z 761.457,A -85,B 0,C 180,E1 -18180,E2 -18180} C_VEL
LIN {X 0,Y 261.109,Z 758.936,A -85,B 0,C 180,E1 -18182.314,E2 -18182.314} C_VEL
LIN {X 0,Y 261.147,Z 755.364,A -85,B 0,C 180,E1 -18184.631,E2 -18184.631} C_VEL
LIN {X 0,Y 261.393,Z 750.644,A -85,B 0,C 180,E1 -18186.949,E2 -18186.949} C_VEL
LIN {X 0,Y 261.795,Z 743.528,A -85,B 0,C 180,E1 -18189.659,E2 -18189.659} C_VEL
LIN {X 0,Y 262.366,Z 735.79,A -85,B 0,C 180,E1 -18191.982,E2 -18191.982} C_VEL
LIN {X 0,Y 263.307,Z 726.274,A -85,B 0,C 180,E1 -18194.294,E2 -18194.294} C_VEL
LIN {X 0,Y 264.053,Z 716.901,A -85,B 0,C 180,E1 -18196.166,E2 -18196.166} C_VEL
LIN {X 0,Y 265.273,Z 706.056,A -85,B 0,C 180,E1 -18197.937,E2 -18197.937} C_VEL
LIN {X 0,Y 266.539,Z 693.093,A -85,B 0,C 180,E1 -18199.645,E2 -18199.645} C_VEL
LIN {X 0,Y 267.599,Z 680.338,A -85,B 0,C 180,E1 -18200.967,E2 -18200.967} C_VEL
LIN {X 0,Y 268.631,Z 666.249,A -85,B 0,C 180,E1 -18202.091,E2 -18202.091} C_VEL
LIN {X 0,Y 269.488,Z 651.394,A -85,B 0,C 180,E1 -18202.927,E2 -18202.927} C_VEL
LIN {X 0,Y 273.067,Z 579.165,A -85,B 0,C 180,E1 -18205.947,E2 -18205.947} C_VEL
LIN {X 0,Y 269.581,Z 548.304,A -85,B 0,C 180,E1 -18207.497,E2 -18207.497} C_VEL
LIN {X 0,Y 268.842,Z 538.437,A -85,B 0,C 180,E1 -18208.007,E2 -18208.007} C_VEL
LIN {X 0,Y 269.557,Z 533.828,A -85,B 0,C 180,E1 -18209.266,E2 -18209.266} C_VEL
LIN {X 0,Y 269.064,Z 529.759,A -85,B 0,C 180,E1 -18210.461,E2 -18210.461} C_VEL
LIN {X 0,Y 265.941,Z 515.121,A -85,B 0,C 180,E1 -18214.991,E2 -18214.991} C_VEL
LIN {X 0,Y 263.17,Z 502.824,A -85,B 0,C 180,E1 -18219.025,E2 -18219.025} C_VEL
LIN {X 0,Y 263.131,Z 502.833,A -85,B 0,C 180,E1 -18221.892,E2 -18221.892} C_VEL
LIN {X 0,Y 263.125,Z 502.833,A -85,B 0,C 180,E1 -18226.15,E2 -18226.15} C_VEL
LIN {X 0,Y 263.107,Z 502.835,A -85,B 0,C 180,E1 -18230.127,E2 -18230.127} C_VEL
LIN {X 0,Y 263.164,Z 502.827,A -85,B 0,C 180,E1 -18234.018,E2 -18234.018} C_VEL
LIN {X 0,Y 263.135,Z 502.833,A -85,B 0,C 180,E1 -18237.712,E2 -18237.712} C_VEL
LIN {X 0,Y 263.203,Z 502.824,A -85,B 0,C 180,E1 -18241.783,E2 -18241.783} C_VEL
LIN {X 0,Y 263.227,Z 502.819,A -85,B 0,C 180,E1 -18245.2,E2 -18245.2} C_VEL
LIN {X 0,Y 263.265,Z 502.817,A -85,B 0,C 180,E1 -18249.693,E2 -18249.693} C_VEL
LIN {X 0,Y 263.352,Z 502.802,A -85,B 0,C 180,E1 -18254.522,E2 -18254.522} C_VEL
LIN {X 0,Y 263.375,Z 502.803,A -85,B 0,C 180,E1 -18259.234,E2 -18259.234} C_VEL
LIN {X 0,Y 263.575,Z 502.774,A -85,B 0,C 180,E1 -18262.338,E2 -18262.338} C_VEL
LIN {X 0,Y 263.756,Z 502.752,A -85,B 0,C 180,E1 -18268.473,E2 -18268.473} C_VEL
LIN {X 0,Y 263.754,Z 502.757,A -85,B 0,C 180,E1 -18271.527,E2 -18271.527} C_VEL
LIN {X 0,Y 263.574,Z 502.776,A -85,B 0,C 180,E1 -18277.662,E2 -18277.662} C_VEL
LIN {X 0,Y 263.375,Z 502.8,A -85,B 0,C 180,E1 -18280.766,E2 -18280.766} C_VEL
LIN {X 0,Y 263.352,Z 502.806,A -85,B 0,C 180,E1 -18285.478,E2 -18285.478} C_VEL
LIN {X 0,Y 263.265,Z 502.814,A -85,B 0,C 180,E1 -18290.307,E2 -18290.307} C_VEL
LIN {X 0,Y 263.209,Z 502.824,A -85,B 0,C 180,E1 -18295.291,E2 -18295.291} C_VEL
LIN {X 0,Y 263.166,Z 502.827,A -85,B 0,C 180,E1 -18298.731,E2 -18298.731} C_VEL
LIN {X 0,Y 263.134,Z 502.829,A -85,B 0,C 180,E1 -18302.288,E2 -18302.288} C_VEL
LIN {X 0,Y 263.189,Z 502.824,A -85,B 0,C 180,E1 -18305.978,E2 -18305.978} C_VEL
LIN {X 0,Y 263.116,Z 502.833,A -85,B 0,C 180,E1 -18309.871,E2 -18309.871} C_VEL
LIN {X 0,Y 263.129,Z 502.831,A -85,B 0,C 180,E1 -18313.983,E2 -18313.983} C_VEL
LIN {X 0,Y 263.126,Z 502.831,A -85,B 0,C 180,E1 -18318.406,E2 -18318.406} C_VEL
LIN {X 0,Y 263.184,Z 502.828,A -85,B 0,C 180,E1 -18323.237,E2 -18323.237} C_VEL
LIN {X 0,Y 263.227,Z 502.995,A -85,B 0,C 180,E1 -18323.979,E2 -18323.979} C_VEL
LIN {X 0,Y 266.934,Z 518.988,A -85,B 0,C 180,E1 -18327.816,E2 -18327.816} C_VEL
LIN {X 0,Y 269.828,Z 532.589,A -85,B 0,C 180,E1 -18330.98,E2 -18330.98} C_VEL
LIN {X 0,Y 269.218,Z 540.864,A -85,B 0,C 180,E1 -18332.728,E2 -18332.728} C_VEL
LIN {X 0,Y 268.359,Z 550.304,A -85,B 0,C 180,E1 -18334.684,E2 -18334.684} C_VEL
LIN {X 0,Y 270.352,Z 572.412,A -85,B 0,C 180,E1 -18335.717,E2 -18335.717} C_VEL
LIN {X 0,Y 271.393,Z 581.069,A -85,B 0,C 180,E1 -18336.128,E2 -18336.128} C_VEL
LIN {X 0,Y 268.067,Z 661.675,A -85,B 0,C 180,E1 -18339.422,E2 -18339.422} C_VEL
